// SIMATIC S7-200 SMART project (STEP 7-Micro/WIN SMART), CPU ST40

SYMBOL_TABLE USER1
Spa_vidé         V102.0   // Spa sans eau pour nettoyage
Compteur0        C0       // Compteur temps Brome
Compteur1        C1       // Compteur cycle filtration HORS usage spa
Compteur2        C2
Compteur3        C3       // Compteur cycle logo BROME
Compteur4        C4       // Compteur jours vérif brome
Bp_Dde_Jets      I0.0     // M/A jets
Bp_Dde_Air       I0.1     // M/A Turbine
Bp_Dde_Ecl       I0.2     // M/A Eclairage
Bp_Dde_Heater    I0.3     // M/A Chauffage=> Non utilisé depuis SPA
Bp_Mode_Hiver    I0.4     // Si=1 alors 1 cycle/jour
Filtration_Forcée I0.5     // Filtration forcée
Filtration_Auto  I0.6     // Filtration en auto
Bp_Arrêt         I0.7     // Arrêt des pompes
Symbol_140       M0.1     // Etat_Air
Bit_1            M1.0     // Forçage à 1
Symbol_28        M2.0     // ModBUS démarré
Symbol_25        M2.1     // carte n°1 ok
Symbol_26        M2.2     // carte n°2 ok
Symbol_27        M2.3     // carte n°3 ok
Symbol_85        M2.4     // carte n°4 ok
Bascule_SR_Jets  M10.0    // M/A jets
Symbol_49        M10.1    // Etat_Air
Bascule_SR_Air   M11.0    // M/A turbine
Bascule_SR_Ecl   M12.0    // M/A eclairage
Symbol_29        MB5      // Etat_Air
Symbol_83        MB10     // Etat_Air
Valeur_jets      MB16
Valeur_air       MB17
valeur_pac       MB18
Valeur_tampon    MB19
Pompe_Jets       Q0.0     // M/A Jets pompe
Pompe_Air        Q0.1     // M/A Turbine
Relais_Ecl       Q0.2     // M/A Eclairage
Relais_PAC       Q0.3     // M/A Pompe à chaleur SPA
Pompe_Filtration Q0.4     // M/A Pompe à filtration
Vanne_Remplissage Q0.5     // M/A Vanne remplissage
Fan_SSR          Q0.6     // Ventilateurs relais SSR et coffret
Led_Jets         Q1.0     // Led Bp Jets +5vdc
Led_Air          Q1.1     // Led Bp Air +5vdc
Led_Ecl          Q1.2     // Led Bp Ecl +5vdc
Led_Heat         Q1.3     // Led Bp Heat +5vdc
Led_Arret        Q1.4     // Led Bp Arrêt +5vdc
Led_Hiver        Q1.5     // Led Mode Hiver
TimerJets        T37      // Tempo jets 30 min
TimerAir         T38      // Tempo jets 30 min
TimerFilt        T39      // Tempo 54min
TimerCyc1        T40      // Tempo 54min
TimerCyc2        T41      // Tempo 54min
TimerCycFilt     T42
Bit_1Hz          T45
Symbol_45        T48      // Etat_Air
Bit_2Hz          T50
Symbol_137       T51      // Etat_Air
Symbol_134       T52      // Etat_Air
Symbol_44        T53      // Etat_Air
TimerRstTpsPompJets T54      // Timer reset tps marche pompe jets
TimerFillSpa     T55      // Timer Remplissage Spa
TimerCarte7      T56      // TimerCycleModbus carte7
TimerCarte6      T57      // TimerCycleModbus carte6
TimerCarte5      T58      // TimerCycleModbus carte5
TimerCycleModbus T59      // TimerCycleModbus
TimerCarte1      T60      // TimerCycleModbus carte1
TimerCarte2      T61      // TimerCycleModbus carte2
TimerCarte3      T62      // TimerCycleModbus carte3
TimerCarte4      T63      // TimerCycleModbus carte4
TimerCycleRS485  T255     // Temporisation cartes RS485
Symbol_2         V10.0    // Etat_Air
Symbol_3         V10.1    // Etat_Air
Symbol_8         V10.2    // Etat_Air
Symbol_0         V11.0    // Demande Air
Symbol_1         V11.1    // Etat_Air
Symbol_7         V11.2    // Etat_Air
Symbol_5         V12.0    // Etat_Air
Symbol_4         V12.1    // Etat_Air
Symbol_6         V12.2    // Etat_Air
DiminuerTauxpH   V51.1
AugmenterTauxpH  V51.2
pHOk             V51.3
Symbol_19        V70.0    // Etat_Air
Symbol_90        V101.0   // Etat_Air
Symbol_91        V201.0   // Etat_Air
BromeLogo        V702.0   // Demande vérification Brome
Symbol_88        V1220.0  // Etat_Air
Symbol_89        V1220.1  // Etat_Air
AckDef           V1510.0  // Effacement des défauts
ResetTpsPompeJets V1510.1  // RàZ du totaliseur de la pompe jets
Symbol_62        V1510.2  // Etat_Air
Symbol_135       V1510.3  // Etat_Air
Symbol_136       V1510.4  // Etat_Air
Symbol_138       V1510.5  // Etat_Air
ResetDéfBrome    V1510.6  // Etat_Air
CorrectionpH     V1799.3  // 1 cycle de correction du pH
Symbol_142       V6000.1  // Etat_Air
Symbol_143       V6000.2  // Etat_Air
Symbol_144       V6000.3  // Etat_Air
Symbol_145       V6000.4  // Etat_Air
Symbol_146       V6000.5  // Etat_Air
Symbol_39        VB0      // Etat_Air
Symbol_40        VB1      // Etat_Air
Symbol_38        VB2      // Etat_Air
Symbol_41        VB3      // Etat_Air
Symbol_56        VB4      // Etat_Air
Symbol_96        VB5      // Etat_Air
Symbol_9         VB15     // Etat_Air
Fond_écran_HMI   VB15
Symbol_11        VB100    // Etat_Air
Symbol_12        VB200    // Etat_Air
Symbol_48        VB500    // Etat_Air
EtatFiltration   VB600    // Etat filtration à sable/cartouche
Symbol_20        VB700    // Etat_Air
Symbol_13        VB1100   // Etat_Air
Symbol_51        VB1200   // Etat_Air
Symbol_92        VB1202   // Etat_Air
Symbol_74        VB1300   // Etat_Air
Symbol_14        VB1400   // Etat_Air
Symbol_93        VB1500   // Etat_Air
Symbol_141       VB1510   // Etat_Air
SensRotationPump VB1710   // 0: sens CW / 1: sens CCW
AccelRotationPump VB1711   // Accélération moteur pompe
Symbol_50        VB2000   // Etat_Air
Symbol_100       VB3000   // Etat_Air
Symbol_21        VD1000   // Etat_Air
NbreTrPump       VD1714   // Nombre tours pompe: 1tr=25600pts
VolumeInjection  VD1780   // Nombre tours injection
NbreTourPompeIhm VD1784   // Nombre tour pompe en manu
Tps_Mar_Pomp_Jets VD3000   // Tps_Mar_Pomp_Jets
Symbol_35        VD3004   // Etat_Air
Symbol_101       VD3008   // Etat_Air
Tps_Mar_Pomp_Air VD3010   // Tps_Mar_Pomp_Air
Symbol_103       VD3012   // Etat_Air
Symbol_15        VD3016   // Etat_Air
Tps_Mar_Pomp_Ecl VD3020   // Tps_Mar_Pomp_Ecl
Symbol_82        VD3028   // Etat_Air
Tps_Mar_Pomp_Pac VD3030   // Tps_Mar_Pomp_Pac
Symbol_63        VD3032   // Etat_Air
Symbol_64        VD3036   // Etat_Air
Tps_Mar_Pomp_Filt VD3040   // Tps_Mar_Pomp_Filt
Symbol_79        VD3044   // Etat_Air
Symbol_81        VD3048   // Etat_Air
Symbol_97        VD3052   // Etat_Air
Symbol_47        VD3100   // Etat_Air
Symbol_16        VD3104   // Etat_Air
Symbol_17        VD3108   // Etat_Air
Symbol_18        VD3112   // Etat_Air
Symbol_133       VD3116   // Etat_Air
Symbol_98        VD3120   // Etat_Air
Symbol_99        VD3124   // Etat_Air
Symbol_102       VD3128   // Etat_Air
Symbol_105       VD3132   // Etat_Air
Symbol_106       VD3136   // Etat_Air
Symbol_107       VD3140   // Etat_Air
Symbol_108       VD3144   // Etat_Air
Symbol_109       VD3148   // Etat_Air
Symbol_110       VD3152   // Etat_Air
Symbol_60        VD3200   // Etat_Air
Symbol_61        VD3300   // Etat_Air
Symbol_111       VD3312   // Etat_Air
Symbol_112       VD3316   // Etat_Air
Symbol_113       VD3320   // Etat_Air
Symbol_114       VD3324   // Etat_Air
Symbol_115       VD3328   // Etat_Air
Symbol_116       VD3332   // Etat_Air
Symbol_117       VD3336   // Etat_Air
Symbol_118       VD3340   // Etat_Air
Symbol_119       VD3344   // Etat_Air
Symbol_120       VD3348   // Etat_Air
Symbol_121       VD3352   // Etat_Air
Symbol_65        VD3400   // Etat_Air
Symbol_122       VD3412   // Etat_Air
Symbol_123       VD3416   // Etat_Air
Symbol_124       VD3420   // Etat_Air
Symbol_125       VD3424   // Etat_Air
Symbol_126       VD3428   // Etat_Air
Symbol_127       VD3432   // Etat_Air
Symbol_128       VD3436   // Etat_Air
Symbol_129       VD3440   // Etat_Air
Symbol_130       VD3444   // Etat_Air
Symbol_131       VD3448   // Etat_Air
Symbol_132       VD3452   // Etat_Air
Symbol_10        VD30012  // Etat_Air
Symbol_77        VD30444  //
NbreCycleFilt    VW7      // nombre cycle filtration par jour
LimiteFiltrationJour VW120    // LimiteFiltrationJour
Symbol_80        VW140    // Etat_Air
Symbol_78        VW150    // Etat_Air
Symbol_24        VW1000   // Temp_Eau
Symbol_30        VW1002   // Temp_Jets
Symbol_31        VW1004   // Temp_Air
Symbol_32        VW1006   // Temp_Filt
Symbol_33        VW1008   // Etat_Air
Symbol_34        VW1010   // Etat_Air
Symbol_37        VW1012   // Etat_Air
Symbol_36        VW1014   // Etat_Air
Symbol_43        VW1020   // Etat_Air
Symbol_46        VW1022   // Etat_Air
Symbol_58        VW1024   // Etat_Air
Symbol_59        VW1026   // Etat_Air
TempératureEau   VW1100   // Température Eau
Symbol_57        VW1102   // Température moteur Jets
Symbol_66        VW1104   // Température moteur Air
Symbol_67        VW1106   // Température moteur Filtration
Symbol_68        VW1108   //
Symbol_69        VW1110   //
Symbol_70        VW1112   //
Symbol_71        VW1114   //
Symbol_72        VW1120   //
Symbol_73        VW1122   //
Symbol_54        VW1200   // pH de l'eau
TauxpHBassin     VW1202   // Température de l'eau (pas utilisée)
LimitPhBas       VW1210   // Limite haute du pH
LimitPhHaut      VW1212   // Limite basse du pH
Symbol_75        VW1300   //
Symbol_76        VW1302   //
Symbol_86        VW1400   //
Symbol_87        VW1402   //
Symbol_94        VW1500   // Etat_Air
Symbol_95        VW1502   // Etat_Air
Demande_Remplissage_Spa VW1520   // Demande_Remplissage
VitesseRotationPump VW1712   // vitesse rotation pompe
TpsSurveillanceTauxpH VW1720   // Surveillance Taux pH toutes les 3h ou 12h
TpsSurveillancePhHiver VW1740   // TpsSurveillancePhHiver
TpsSurveillancePhEté VW1750   // TpsSurveillancePhEté
VitesseRotationPompe VW1770   // Vitesse rotation pompe pH
NombreTourPompe  VW1784   // Nombre tour pompe par défaut
ValeurInjectionDefaut VW1786   // valeur par défaut pour rester à 7.4
Symbol_52        VW2000   //
Symbol_53        VW2002   //
Symbol_22        VW3000   // Etat_Air
Symbol_104       VW3002   // Etat_Air
Symbol_23        VW3004   // Etat_Air
Symbol_84        VW3304   // Etat_Air
OffsetPh         VW7000   // offset sur sonde pH
OffsetOrp        VW7002   // Offset sonde ORP
END_SYMBOL_TABLE

SYMBOL_TABLE Table 2
PTO3_Status      SMB580   // PTO3 Status
PLS3_Ovr         SM580.6  // PTO3 pipeline overflow/underflow, loading pipeline while full or transferring an empty pipeline: 0=No overflow; 1=Pipeline overflow/underflow
PLS3_Idle        SM580.7  // PTO3 idle: 0 = PTO in progress;1= PTO is idle
PLS3_Ctrl        SMB581   // Monitor and control PTO3 (Pulse Train Output) and PWM3 (Pulse Width Modulation) for Q0.2
PLS3_Cycle_Update SM581.0  // PTO3/PWM3 update the cycle time or frequency value: 0=no update; 1=write new cycle time/frequency
PWM3_PW_Update   SM581.1  // PWM3 update the pulse width value: 0=no update; 1= write new pulse width
PTO3_PC_Update   SM581.2  // PTO3 update the pulse count value: 0=no update; 1= write new pulse count
PWM3_TimeBase    SM581.3  // PWM3 time base: 0=1us/tick, 1=1ms/tick
PLS3_Select      SM581.6  // PTO3/PWM3 mode select: 0=PWM; 1=PTO.
PLS3_Enable      SM581.7  // PTO3/PWM3 enable: 0=disable; 1=enable.
PLS3_Cycle       SMW582   // PWM3 cycle time value (2 to 65,535 units of time base); PTO3 frequency value (1 to 65,535 Hz)
PWM3_PW          SMW584   // PWM3 pulse width value (0 to 65,535 units of time base)
PTO3_PC          SMD586   // PTO3 pulse count value (1 to 2^32 - 1)
PLS3_Abort_AE    SM580.4  // PTO3 profile was aborted due to an add error: 0=no abort; 1=aborted
PLS3_Disable_UC  SM580.5  // PTO3 user manually disabled a PTO profile while it was running: 0=not disabled; 1=manually disabled
PTO3_Operation   SM581.5  // PTO3 select single/multiple segment operation: 0=single; 1=multiple
PTO3_Seg_Num     SMB590   // The currently executing segment number for PTO3's profile
PTO3_Profile_Offset SMW592   // Starting location of PTO3's profile table (byte offset from V0)
HSC0_TYPE        SMB195   // HSC0 type: 0=Count 1=Frequency
HSC0_FREQ_PERIOD SMB196   // HSC0 frequency measuring period: 0=1s 1=100ms 2=10ms
HSC1_TYPE        SMB197   // HSC1 type: 0=Count 1=Frequency
HSC1_FREQ_PERIOD SMB198   // HSC1 frequency measuring period: 0=1s 1=100ms 2=10ms
HSC2_TYPE        SMB199   // HSC2 type: 0=Count 1=Frequency
HSC2_FREQ_PERIOD SMB200   // HSC2 frequency measuring period: 0=1s 1=100ms 2=10ms
HSC3_TYPE        SMB201   // HSC3 type: 0=Count 1=Frequency
HSC3_FREQ_PERIOD SMB202   // HSC3 frequency measuring period: 0=1s 1=100ms 2=10ms
HSC4_TYPE        SMB203   // HSC4 type: 0=Count 1=Frequency
HSC4_FREQ_PERIOD SMB204   // HSC4 frequency measuring period: 0=1s 1=100ms 2=10ms
HSC5_TYPE        SMB205   // HSC5 type: 0=Count 1=Frequency
HSC5_FREQ_PERIOD SMB206   // HSC5 frequency measuring period: 0=1s 1=100ms 2=10ms
END_SYMBOL_TABLE

ORGANIZATION_BLOCK PPAL:OB1
TITLE=COMMENTAIRES DE PROGRAMME
VAR
Etat_Jets:BOOL;	// L0.0 Etat Jets
Sortie_Jets:BOOL;	// L0.1 Pilotage Sortie Jets
Voyant_Jets:BOOL;	// L0.2 Voyant +5vdc Jets
END_VAR
BEGIN
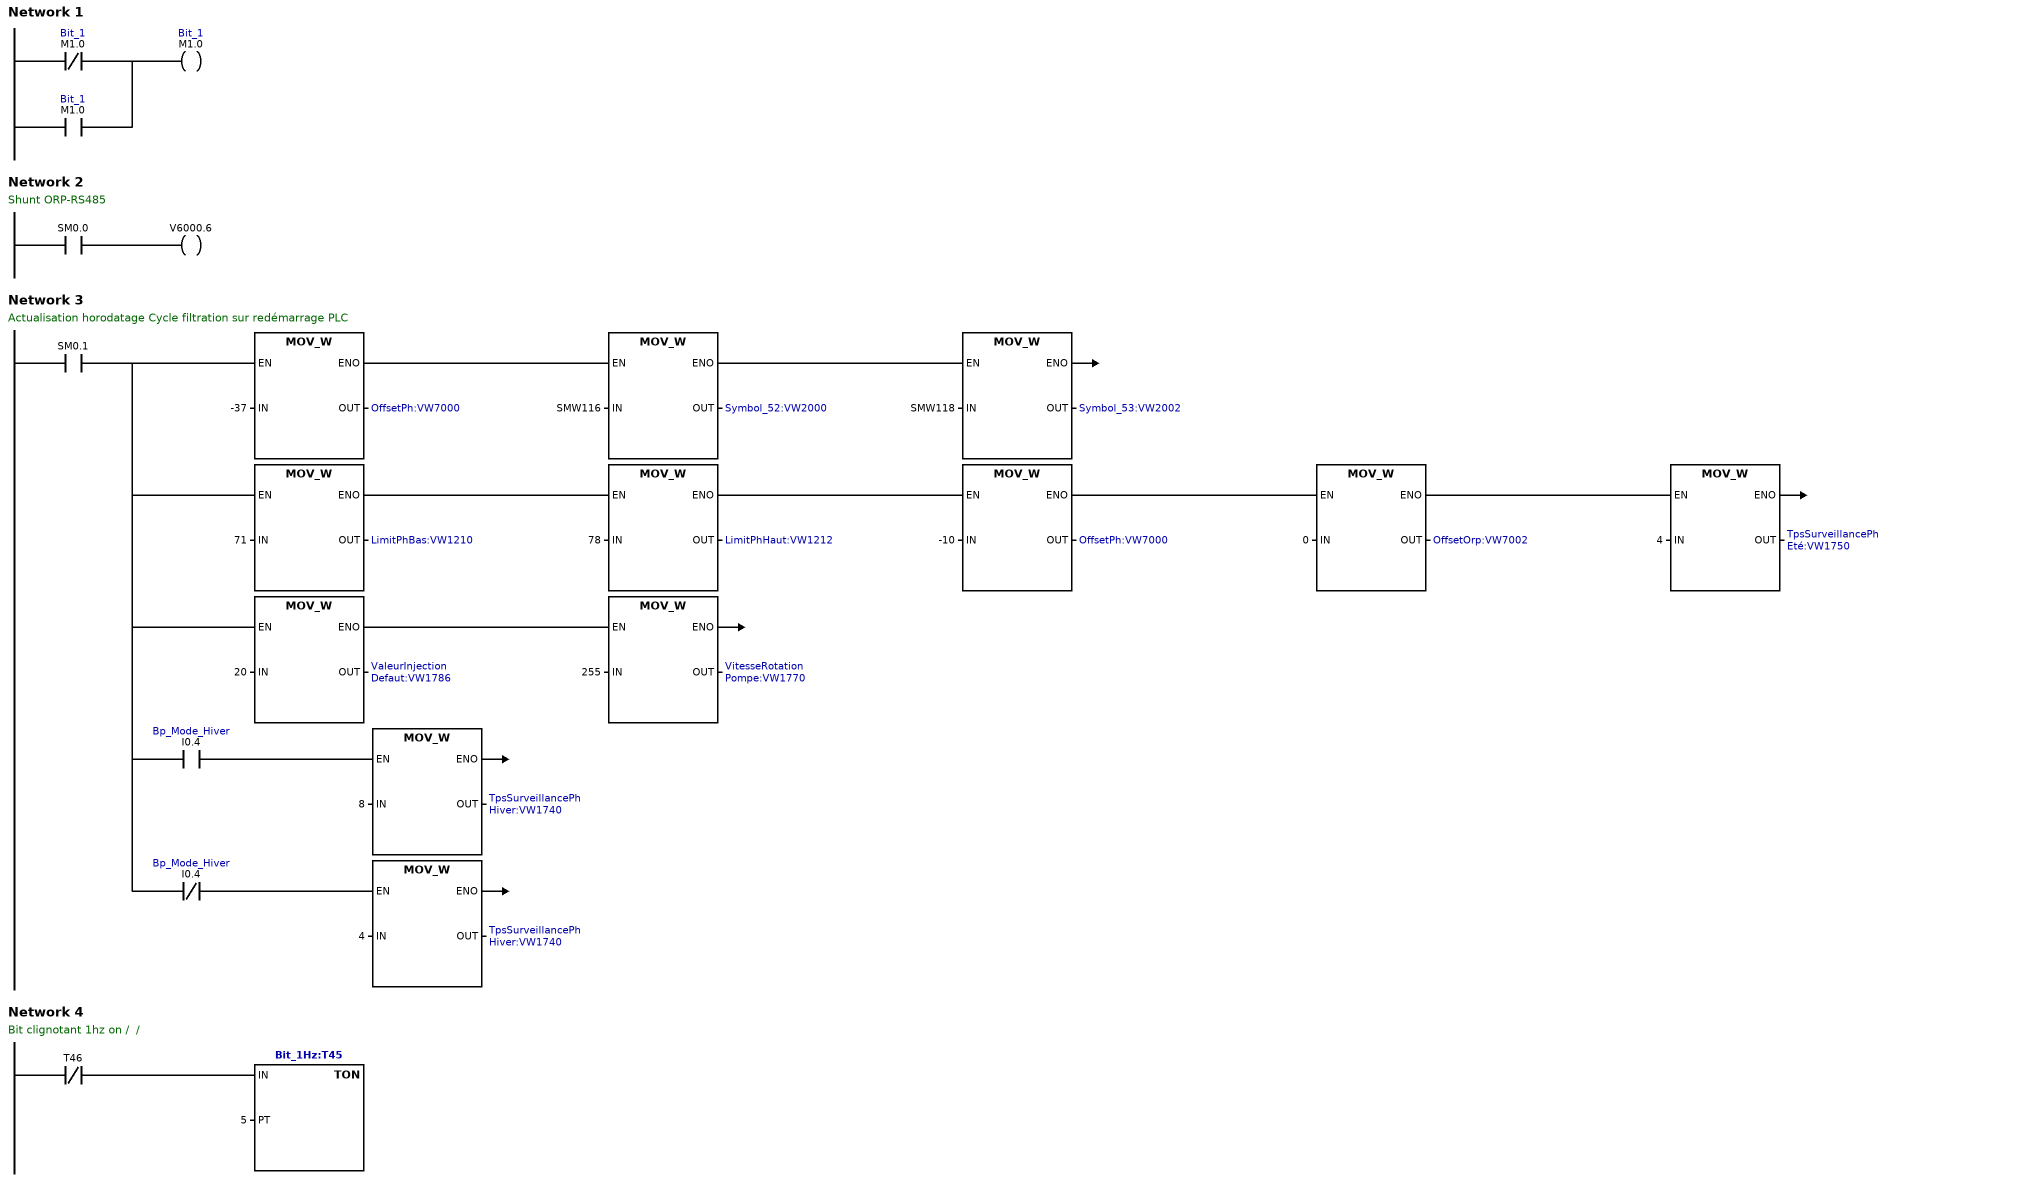
Network 1
LDN    Bit_1:M1.0
O      Bit_1:M1.0
=      Bit_1:M1.0
Network 2
// Shunt ORP-RS485
LD     SM0.0
=      V6000.6
Network 3
// Actualisation horodatage Cycle filtration sur redémarrage PLC
LD     SM0.1
LPS
MOVW   -37, OffsetPh:VW7000
AENO
MOVW   SMW116, Symbol_52:VW2000
AENO
MOVW   SMW118, Symbol_53:VW2002
LRD
MOVW   71, LimitPhBas:VW1210
AENO
MOVW   78, LimitPhHaut:VW1212
AENO
MOVW   -10, OffsetPh:VW7000
AENO
MOVW   0, OffsetOrp:VW7002
AENO
MOVW   4, TpsSurveillancePhEté:VW1750
LRD
MOVW   20, ValeurInjectionDefaut:VW1786
AENO
MOVW   255, VitesseRotationPompe:VW1770
LRD
A      Bp_Mode_Hiver:I0.4
MOVW   8, TpsSurveillancePhHiver:VW1740
LPP
AN     Bp_Mode_Hiver:I0.4
MOVW   4, TpsSurveillancePhHiver:VW1740
Network 4
// Bit clignotant 1hz on
// 
// 
LDN    T46
TON    Bit_1Hz:T45, 5
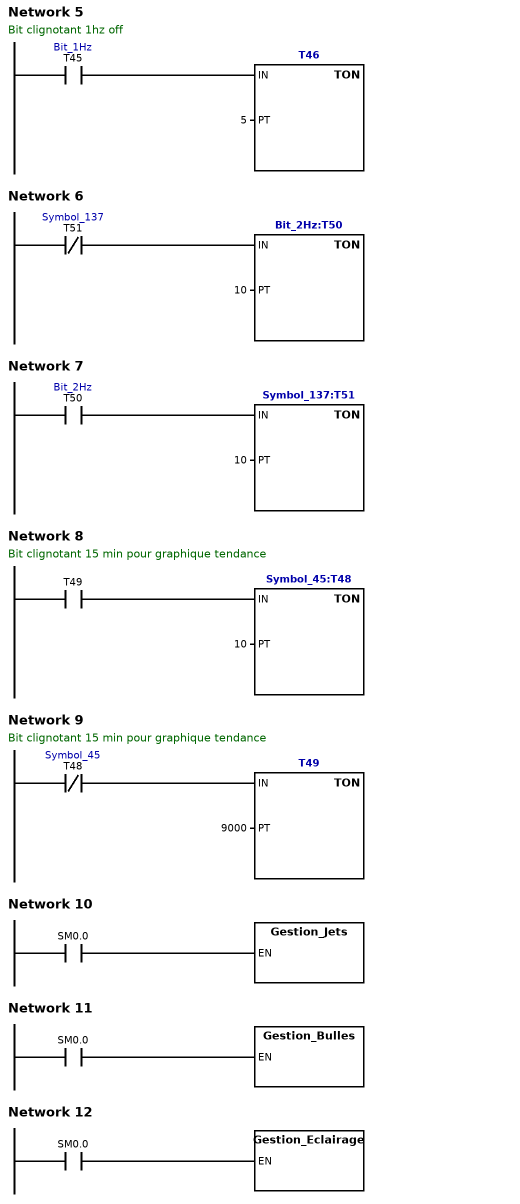
Network 5
// Bit clignotant 1hz off
LD     Bit_1Hz:T45
TON    T46, 5
Network 6
LDN    Symbol_137:T51
TON    Bit_2Hz:T50, 10
Network 7
LD     Bit_2Hz:T50
TON    Symbol_137:T51, 10
Network 8
// Bit clignotant 15 min pour graphique tendance
LD     T49
TON    Symbol_45:T48, 10
Network 9
// Bit clignotant 15 min pour graphique tendance
LDN    Symbol_45:T48
TON    T49, 9000
Network 10
LD     SM0.0
CALL   Gestion_Jets:SBR0
Network 11
LD     SM0.0
CALL   Gestion_Bulles:SBR1
Network 12
LD     SM0.0
CALL   Gestion_Eclairage:SBR2
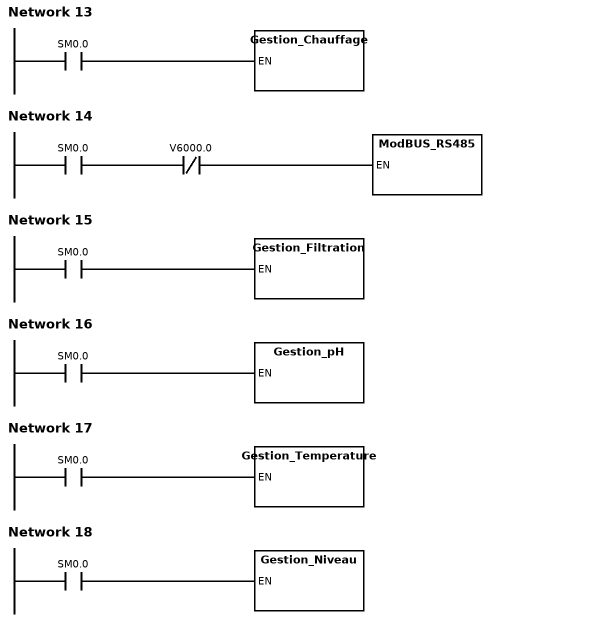
Network 13
LD     SM0.0
CALL   Gestion_Chauffage:SBR3
Network 14
LD     SM0.0
AN     V6000.0
CALL   ModBUS_RS485:SBR5
Network 15
LD     SM0.0
CALL   Gestion_Filtration:SBR7
Network 16
LD     SM0.0
CALL   Gestion_pH:SBR4
Network 17
LD     SM0.0
CALL   Gestion_Temperature:SBR6
Network 18
LD     SM0.0
CALL   Gestion_Niveau:SBR14
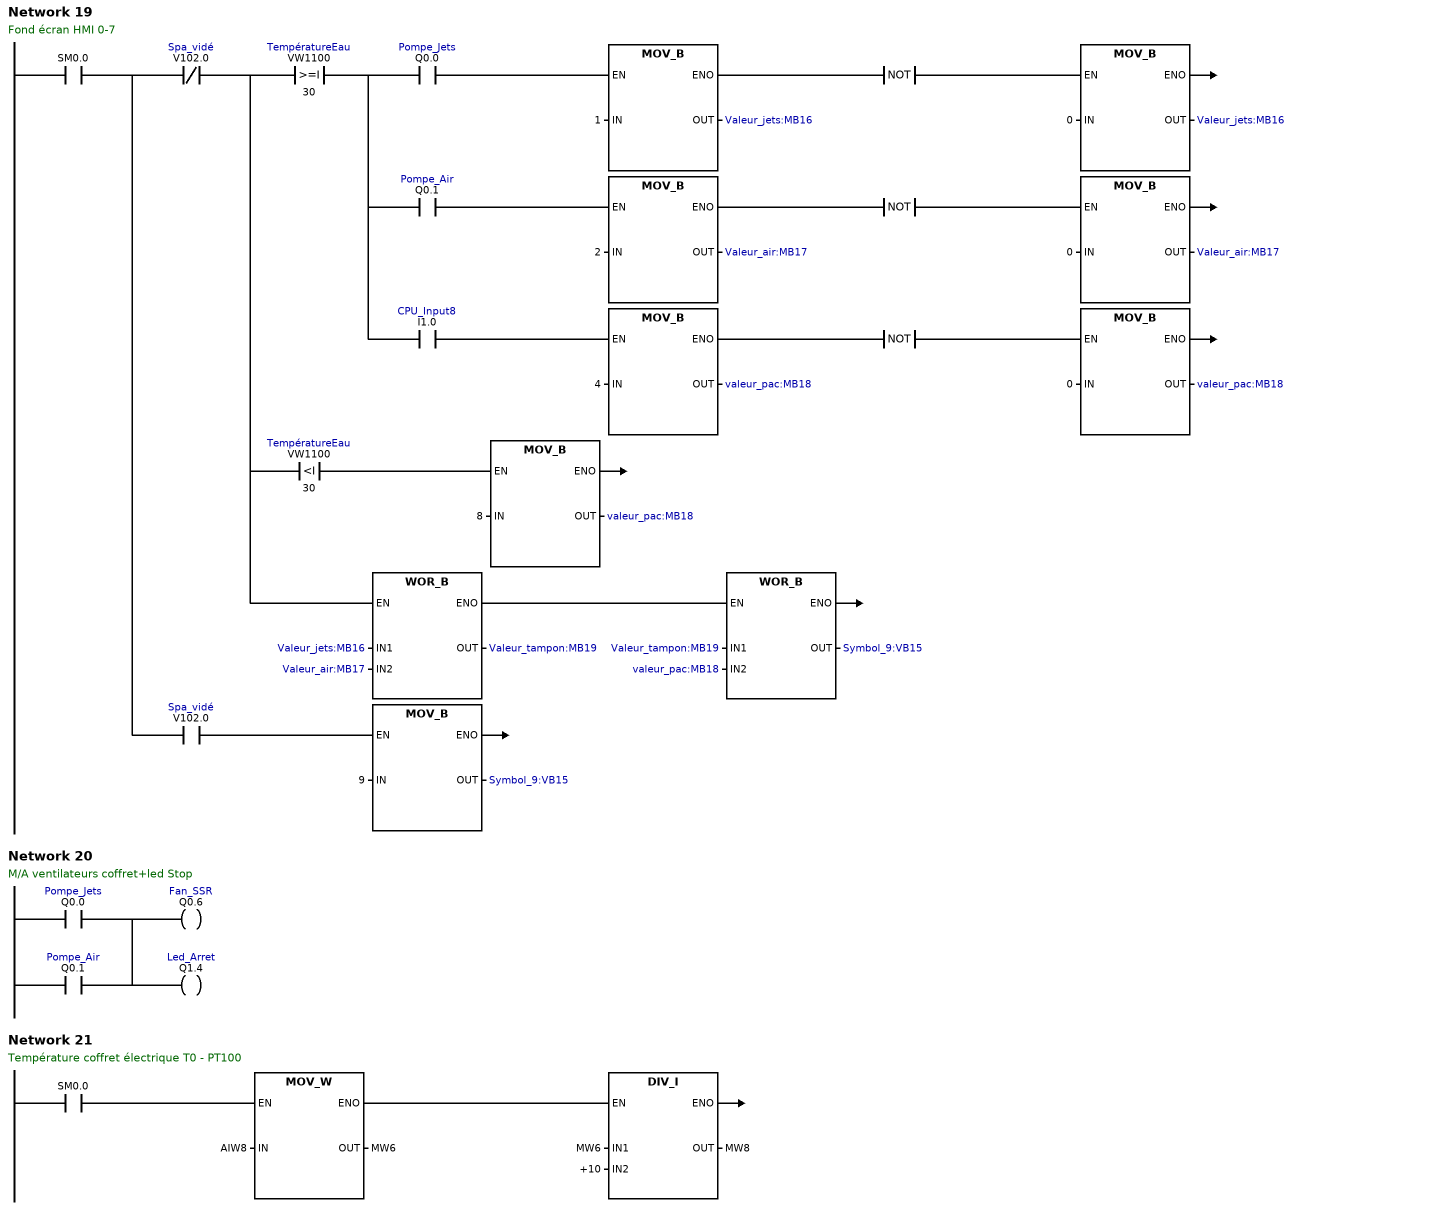
Network 19
// Fond écran HMI 0-7
LD     SM0.0
LPS
AN     Spa_vidé:V102.0
LPS
AW>=   TempératureEau:VW1100, 30
LPS
A      Pompe_Jets:Q0.0
MOVB   1, Valeur_jets:MB16
AENO
NOT
MOVB   0, Valeur_jets:MB16
LRD
A      Pompe_Air:Q0.1
MOVB   2, Valeur_air:MB17
AENO
NOT
MOVB   0, Valeur_air:MB17
LPP
A      CPU_Input8:I1.0
MOVB   4, valeur_pac:MB18
AENO
NOT
MOVB   0, valeur_pac:MB18
LPP
LPS
AW<    TempératureEau:VW1100, 30
MOVB   8, valeur_pac:MB18
LPP
MOVB   Valeur_jets:MB16, Valeur_tampon:MB19
AENO
ORB    Valeur_air:MB17, Valeur_tampon:MB19
AENO
MOVB   Valeur_tampon:MB19, Symbol_9:VB15
ORB    valeur_pac:MB18, Symbol_9:VB15
LPP
A      Spa_vidé:V102.0
MOVB   9, Symbol_9:VB15
Network 20
// M/A ventilateurs coffret+led Stop
LD     Pompe_Jets:Q0.0
O      Pompe_Air:Q0.1
=      Fan_SSR:Q0.6
=      Led_Arret:Q1.4
Network 21
// Température coffret électrique T0 - PT100
LD     SM0.0
MOVW   AIW8, MW6
AENO
MOVW   MW6, MW8
/I     +10, MW8
END_ORGANIZATION_BLOCK

SUBROUTINE_BLOCK Gestion_Jets:SBR0
TITLE=COMMENTAIRES DE SOUS-PROGRAMME
VAR
Etat_Jets:BOOL;	// L0.0 
END_VAR
BEGIN
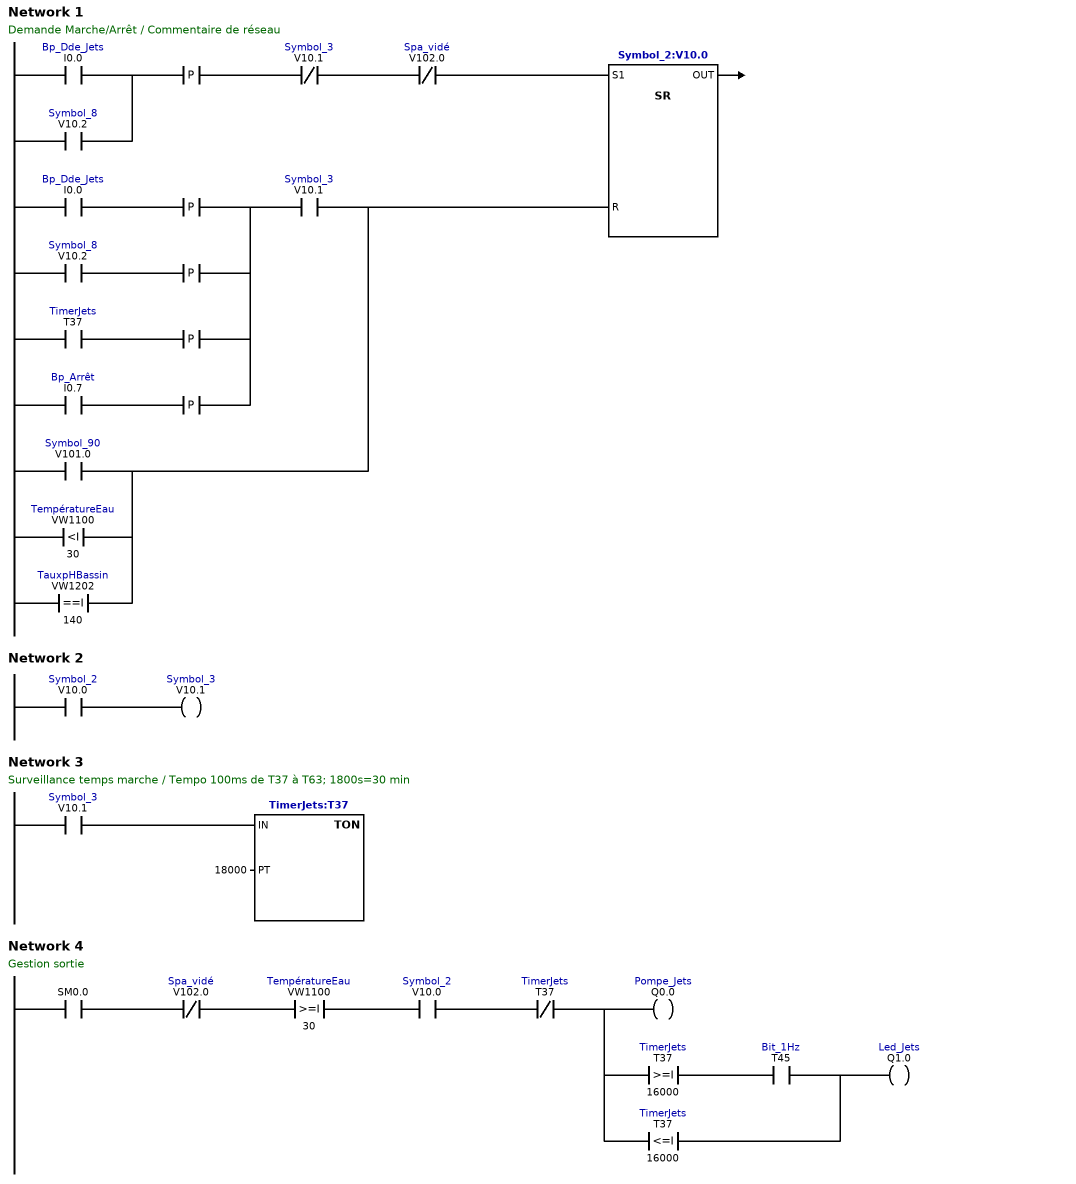
Network 1
// Demande Marche/Arrêt
// Commentaire de réseau
LD     Bp_Dde_Jets:I0.0
O      Symbol_8:V10.2
EU
AN     Symbol_3:V10.1
AN     Spa_vidé:V102.0
LD     Bp_Dde_Jets:I0.0
EU
LD     Symbol_8:V10.2
EU
OLD
LD     TimerJets:T37
EU
OLD
LD     Bp_Arrêt:I0.7
EU
OLD
A      Symbol_3:V10.1
LD     Symbol_90:V101.0
OW<    TempératureEau:VW1100, 30
OW=    TauxpHBassin:VW1202, 140
OLD
NOT
A      Symbol_2:V10.0
OLD
=      Symbol_2:V10.0
Network 2
LD     Symbol_2:V10.0
=      Symbol_3:V10.1
Network 3
// Surveillance temps marche
// Tempo 100ms de T37 à T63; 1800s=30 min
LD     Symbol_3:V10.1
TON    TimerJets:T37, 18000
Network 4
// Gestion sortie
LD     SM0.0
AN     Spa_vidé:V102.0
AW>=   TempératureEau:VW1100, 30
A      Symbol_2:V10.0
AN     TimerJets:T37
=      Pompe_Jets:Q0.0
LDW>=  TimerJets:T37, 16000
A      Bit_1Hz:T45
OW<=   TimerJets:T37, 16000
ALD
=      Led_Jets:Q1.0
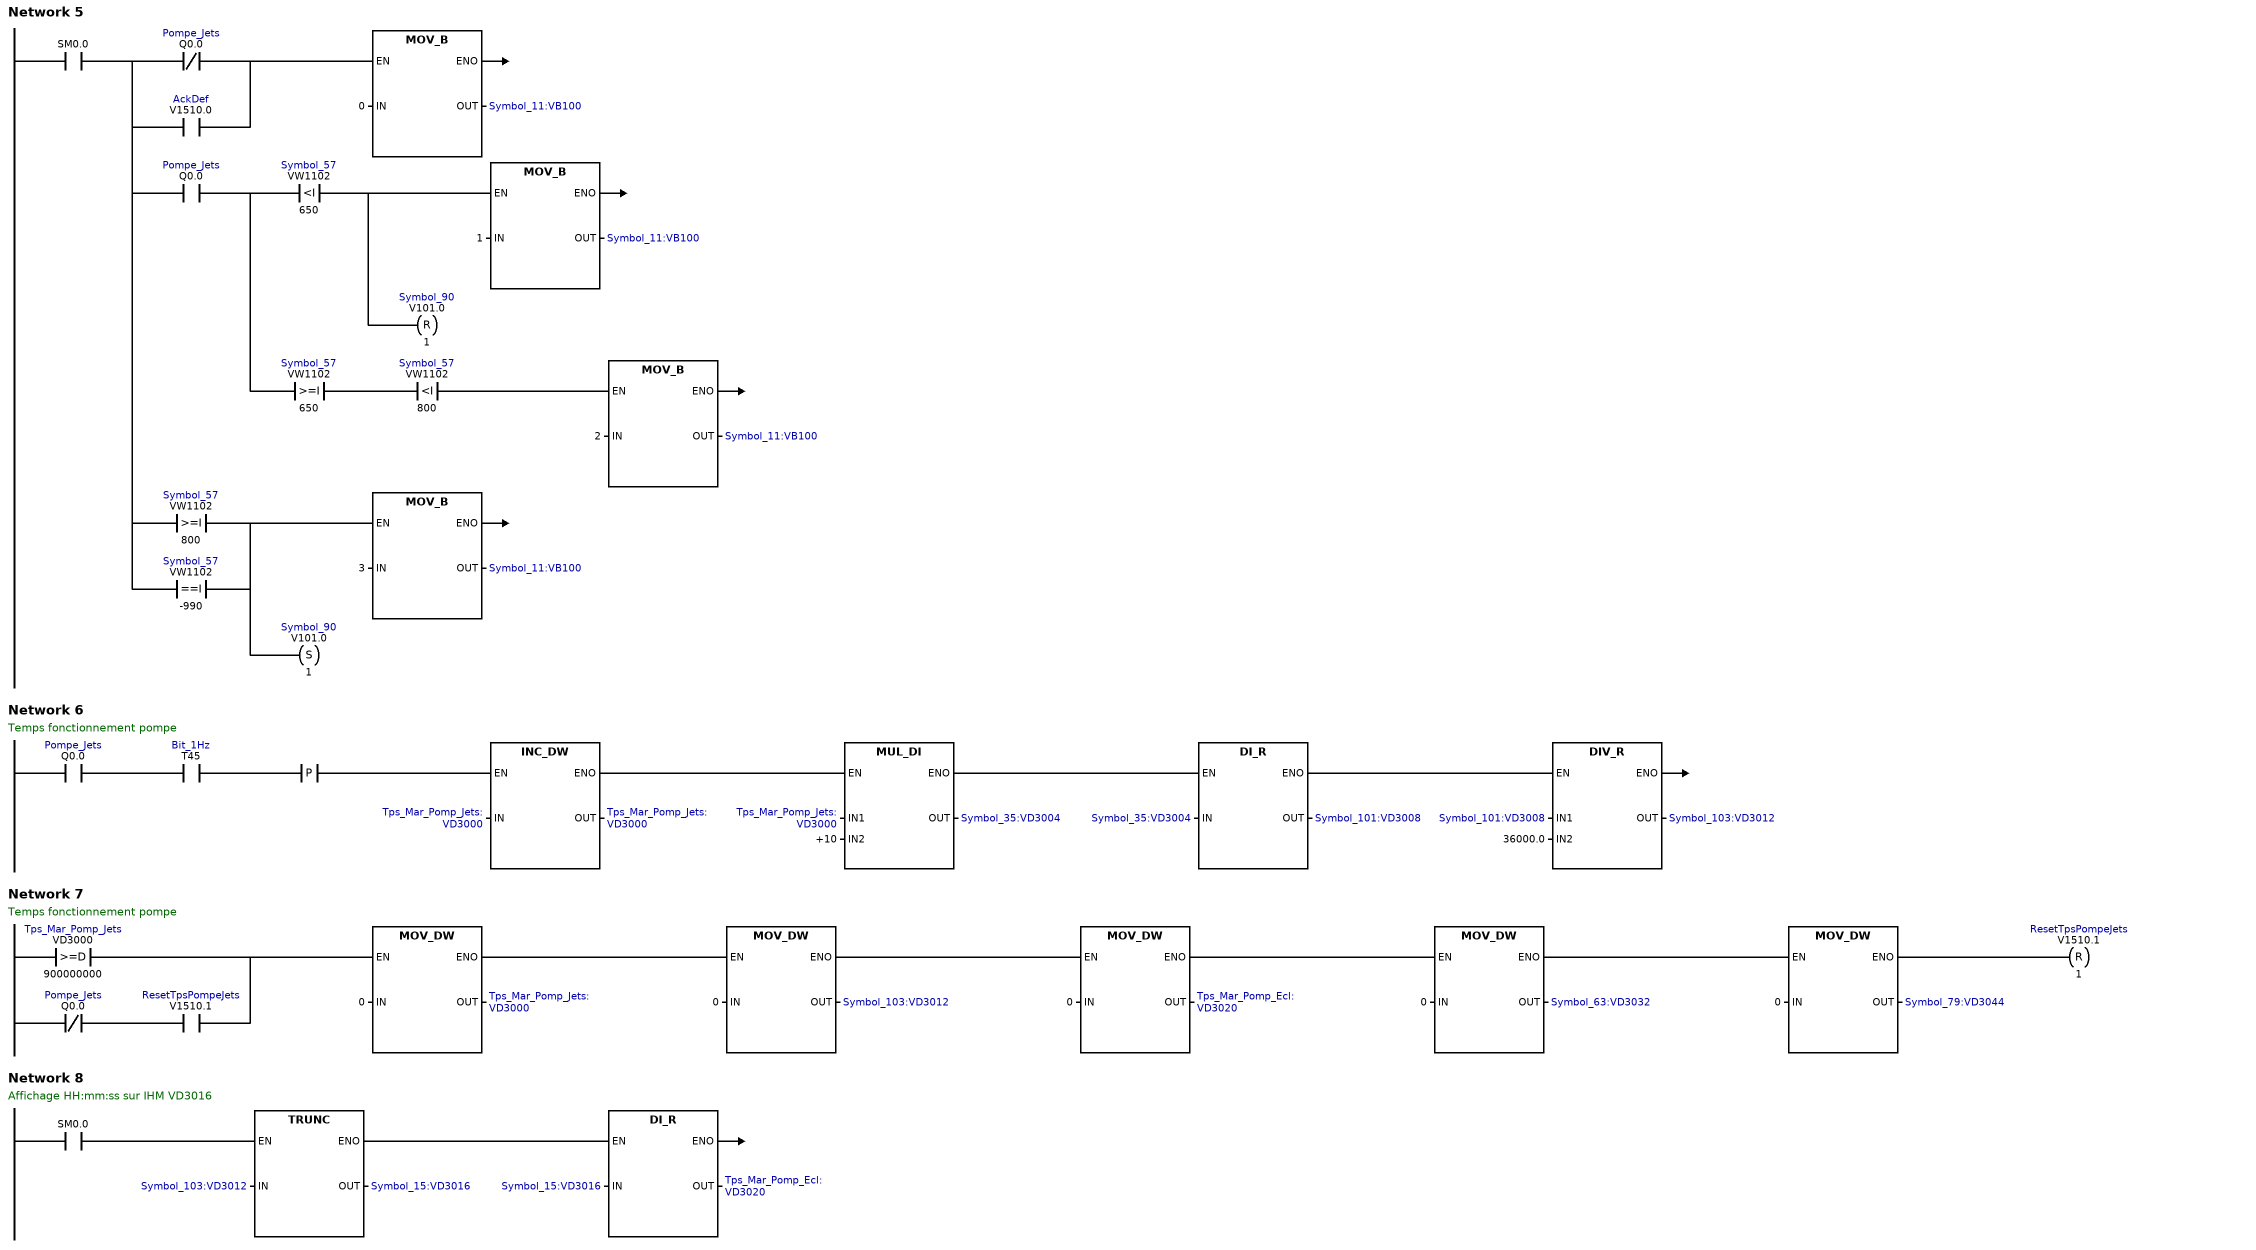
Network 5
LD     SM0.0
LPS
LDN    Pompe_Jets:Q0.0
O      AckDef:V1510.0
ALD
MOVB   0, Symbol_11:VB100
LRD
A      Pompe_Jets:Q0.0
LPS
AW<    Symbol_57:VW1102, 650
MOVB   1, Symbol_11:VB100
R      Symbol_90:V101.0, 1
LPP
AW>=   Symbol_57:VW1102, 650
AW<    Symbol_57:VW1102, 800
MOVB   2, Symbol_11:VB100
LPP
LDW>=  Symbol_57:VW1102, 800
OW=    Symbol_57:VW1102, -990
ALD
MOVB   3, Symbol_11:VB100
S      Symbol_90:V101.0, 1
Network 6
// Temps fonctionnement pompe
LD     Pompe_Jets:Q0.0
A      Bit_1Hz:T45
EU
INCD   Tps_Mar_Pomp_Jets:VD3000
AENO
MOVD   Tps_Mar_Pomp_Jets:VD3000, Symbol_35:VD3004
AENO
*D     +10, Symbol_35:VD3004
AENO
DTR    Symbol_35:VD3004, Symbol_101:VD3008
AENO
MOVR   Symbol_101:VD3008, Symbol_103:VD3012
/R     36000.0, Symbol_103:VD3012
Network 7
// Temps fonctionnement pompe
LDD>=  Tps_Mar_Pomp_Jets:VD3000, 900000000
LDN    Pompe_Jets:Q0.0
A      ResetTpsPompeJets:V1510.1
OLD
MOVD   0, Tps_Mar_Pomp_Jets:VD3000
AENO
MOVD   0, Symbol_103:VD3012
AENO
MOVD   0, Tps_Mar_Pomp_Ecl:VD3020
AENO
MOVD   0, Symbol_63:VD3032
AENO
MOVD   0, Symbol_79:VD3044
AENO
R      ResetTpsPompeJets:V1510.1, 1
Network 8
// Affichage HH:mm:ss sur IHM VD3016
LD     SM0.0
TRUNC  Symbol_103:VD3012, Symbol_15:VD3016
AENO
DTR    Symbol_15:VD3016, Tps_Mar_Pomp_Ecl:VD3020
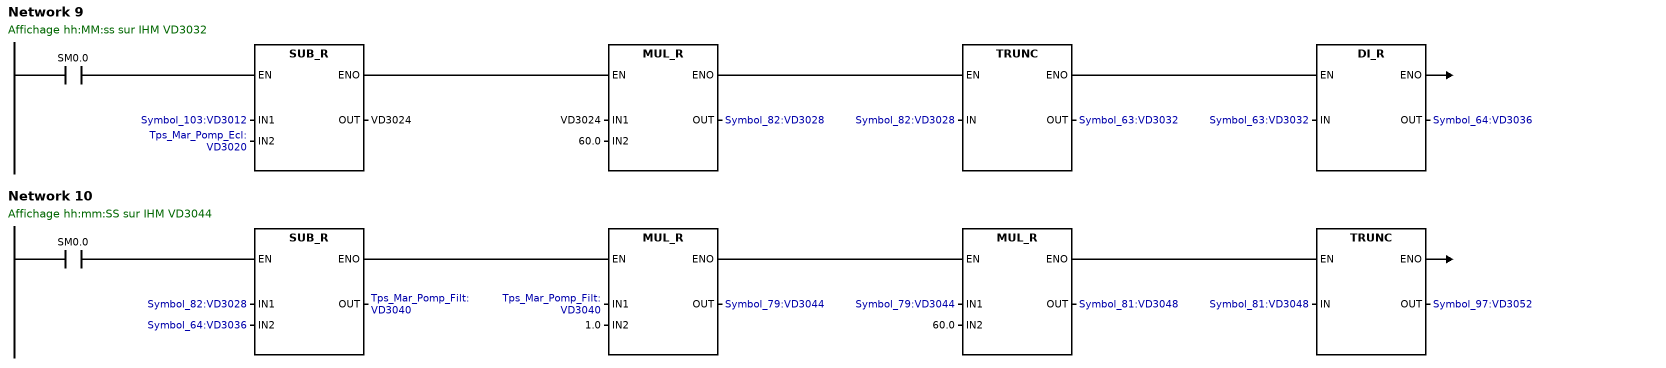
Network 9
// Affichage hh:MM:ss sur IHM VD3032
LD     SM0.0
MOVR   Symbol_103:VD3012, VD3024
AENO
-R     Tps_Mar_Pomp_Ecl:VD3020, VD3024
AENO
MOVR   VD3024, Symbol_82:VD3028
AENO
*R     60.0, Symbol_82:VD3028
AENO
TRUNC  Symbol_82:VD3028, Symbol_63:VD3032
AENO
DTR    Symbol_63:VD3032, Symbol_64:VD3036
Network 10
// Affichage hh:mm:SS sur IHM VD3044
LD     SM0.0
MOVR   Symbol_82:VD3028, Tps_Mar_Pomp_Filt:VD3040
AENO
-R     Symbol_64:VD3036, Tps_Mar_Pomp_Filt:VD3040
AENO
MOVR   Tps_Mar_Pomp_Filt:VD3040, Symbol_79:VD3044
AENO
*R     1.0, Symbol_79:VD3044
AENO
MOVR   Symbol_79:VD3044, Symbol_81:VD3048
AENO
*R     60.0, Symbol_81:VD3048
AENO
TRUNC  Symbol_81:VD3048, Symbol_97:VD3052
END_SUBROUTINE_BLOCK

SUBROUTINE_BLOCK Gestion_Bulles:SBR1
TITLE=COMMENTAIRES DE SOUS-PROGRAMME
VAR
Etat_Air:BOOL;	// L0.0 
END_VAR
BEGIN
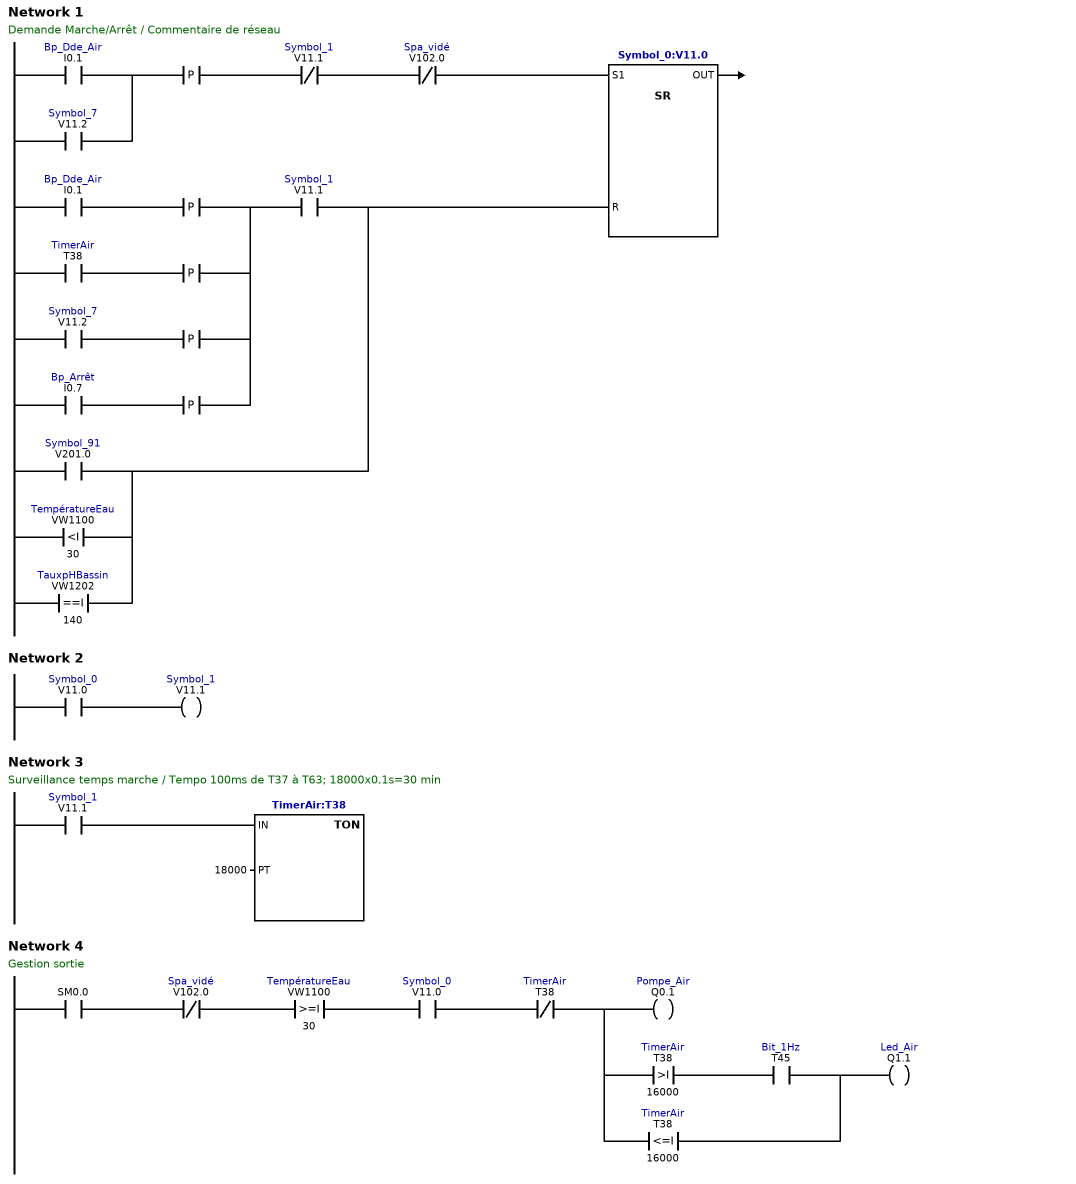
Network 1
// Demande Marche/Arrêt
// Commentaire de réseau
LD     Bp_Dde_Air:I0.1
O      Symbol_7:V11.2
EU
AN     Symbol_1:V11.1
AN     Spa_vidé:V102.0
LD     Bp_Dde_Air:I0.1
EU
LD     TimerAir:T38
EU
OLD
LD     Symbol_7:V11.2
EU
OLD
LD     Bp_Arrêt:I0.7
EU
OLD
A      Symbol_1:V11.1
LD     Symbol_91:V201.0
OW<    TempératureEau:VW1100, 30
OW=    TauxpHBassin:VW1202, 140
OLD
NOT
A      Symbol_0:V11.0
OLD
=      Symbol_0:V11.0
Network 2
LD     Symbol_0:V11.0
=      Symbol_1:V11.1
Network 3
// Surveillance temps marche
// Tempo 100ms de T37 à T63; 18000x0.1s=30 min
LD     Symbol_1:V11.1
TON    TimerAir:T38, 18000
Network 4
// Gestion sortie
LD     SM0.0
AN     Spa_vidé:V102.0
AW>=   TempératureEau:VW1100, 30
A      Symbol_0:V11.0
AN     TimerAir:T38
=      Pompe_Air:Q0.1
LDW>   TimerAir:T38, 16000
A      Bit_1Hz:T45
OW<=   TimerAir:T38, 16000
ALD
=      Led_Air:Q1.1
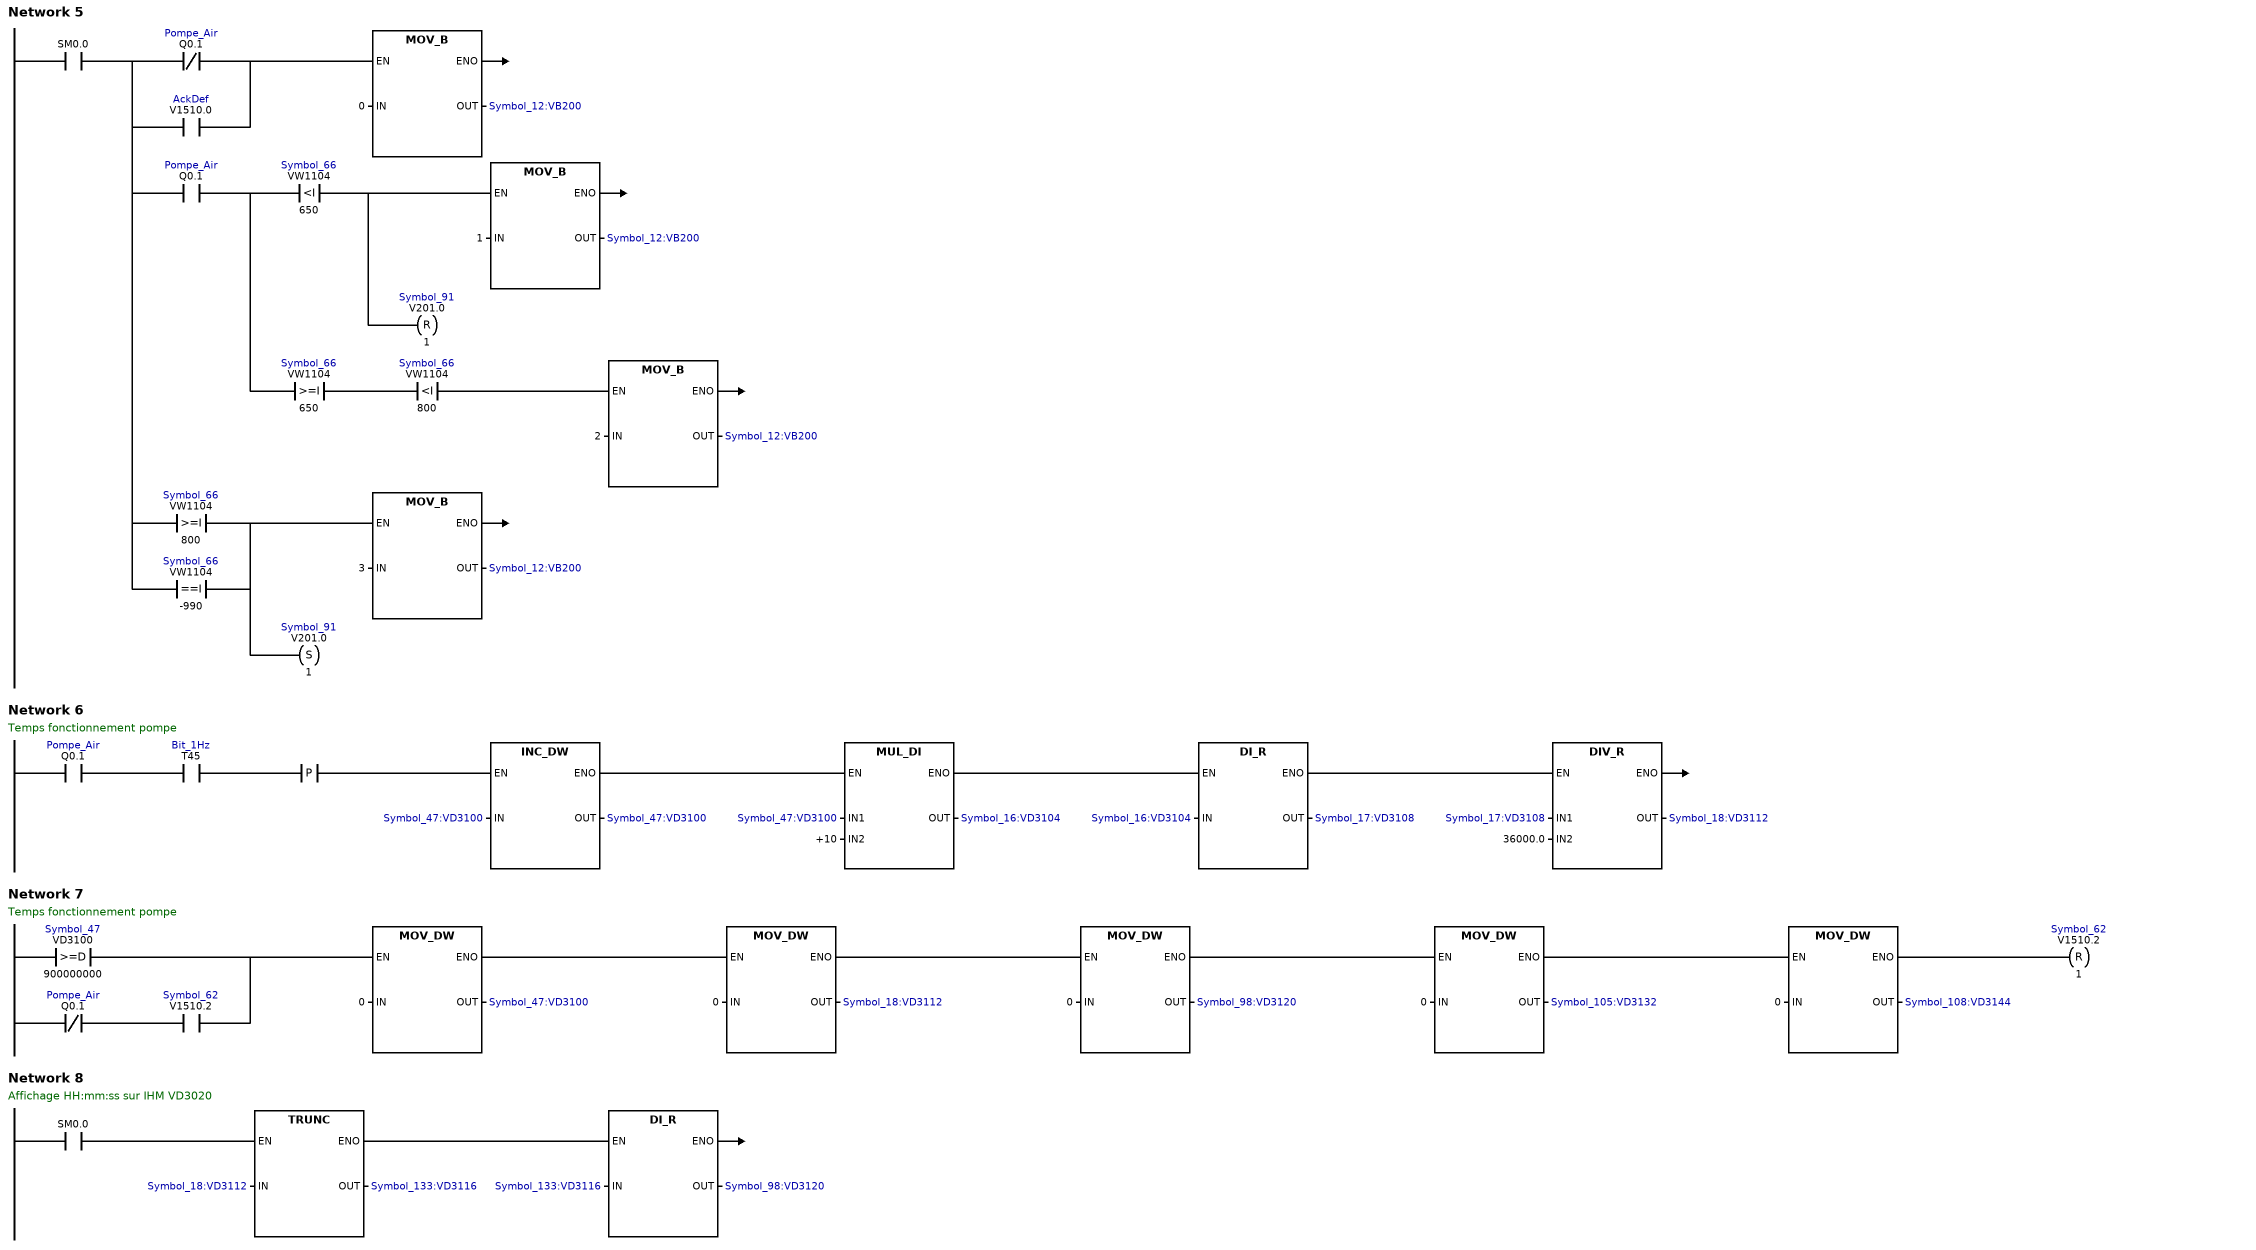
Network 5
LD     SM0.0
LPS
LDN    Pompe_Air:Q0.1
O      AckDef:V1510.0
ALD
MOVB   0, Symbol_12:VB200
LRD
A      Pompe_Air:Q0.1
LPS
AW<    Symbol_66:VW1104, 650
MOVB   1, Symbol_12:VB200
R      Symbol_91:V201.0, 1
LPP
AW>=   Symbol_66:VW1104, 650
AW<    Symbol_66:VW1104, 800
MOVB   2, Symbol_12:VB200
LPP
LDW>=  Symbol_66:VW1104, 800
OW=    Symbol_66:VW1104, -990
ALD
MOVB   3, Symbol_12:VB200
S      Symbol_91:V201.0, 1
Network 6
// Temps fonctionnement pompe
LD     Pompe_Air:Q0.1
A      Bit_1Hz:T45
EU
INCD   Symbol_47:VD3100
AENO
MOVD   Symbol_47:VD3100, Symbol_16:VD3104
AENO
*D     +10, Symbol_16:VD3104
AENO
DTR    Symbol_16:VD3104, Symbol_17:VD3108
AENO
MOVR   Symbol_17:VD3108, Symbol_18:VD3112
/R     36000.0, Symbol_18:VD3112
Network 7
// Temps fonctionnement pompe
LDD>=  Symbol_47:VD3100, 900000000
LDN    Pompe_Air:Q0.1
A      Symbol_62:V1510.2
OLD
MOVD   0, Symbol_47:VD3100
AENO
MOVD   0, Symbol_18:VD3112
AENO
MOVD   0, Symbol_98:VD3120
AENO
MOVD   0, Symbol_105:VD3132
AENO
MOVD   0, Symbol_108:VD3144
AENO
R      Symbol_62:V1510.2, 1
Network 8
// Affichage HH:mm:ss sur IHM VD3020
LD     SM0.0
TRUNC  Symbol_18:VD3112, Symbol_133:VD3116
AENO
DTR    Symbol_133:VD3116, Symbol_98:VD3120
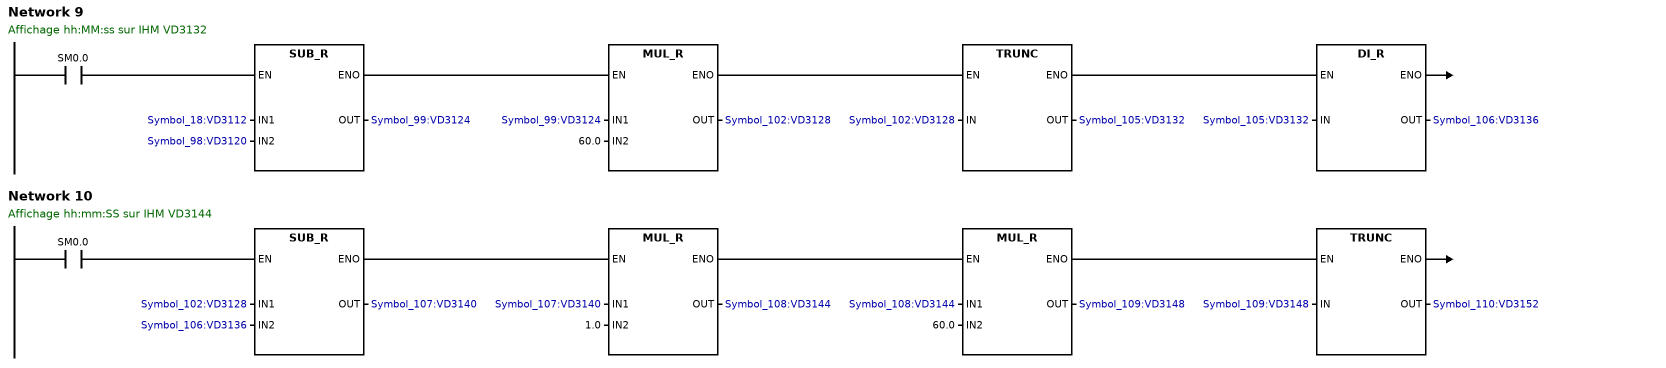
Network 9
// Affichage hh:MM:ss sur IHM VD3132
LD     SM0.0
MOVR   Symbol_18:VD3112, Symbol_99:VD3124
AENO
-R     Symbol_98:VD3120, Symbol_99:VD3124
AENO
MOVR   Symbol_99:VD3124, Symbol_102:VD3128
AENO
*R     60.0, Symbol_102:VD3128
AENO
TRUNC  Symbol_102:VD3128, Symbol_105:VD3132
AENO
DTR    Symbol_105:VD3132, Symbol_106:VD3136
Network 10
// Affichage hh:mm:SS sur IHM VD3144
LD     SM0.0
MOVR   Symbol_102:VD3128, Symbol_107:VD3140
AENO
-R     Symbol_106:VD3136, Symbol_107:VD3140
AENO
MOVR   Symbol_107:VD3140, Symbol_108:VD3144
AENO
*R     1.0, Symbol_108:VD3144
AENO
MOVR   Symbol_108:VD3144, Symbol_109:VD3148
AENO
*R     60.0, Symbol_109:VD3148
AENO
TRUNC  Symbol_109:VD3148, Symbol_110:VD3152
Network 13
// Titre de réseau
// Commentaire de réseau
END_SUBROUTINE_BLOCK

SUBROUTINE_BLOCK Gestion_Eclairage:SBR2
TITLE=COMMENTAIRES DE SOUS-PROGRAMME
VAR
Etat_Ecl:BOOL;	// L0.0 
END_VAR
BEGIN
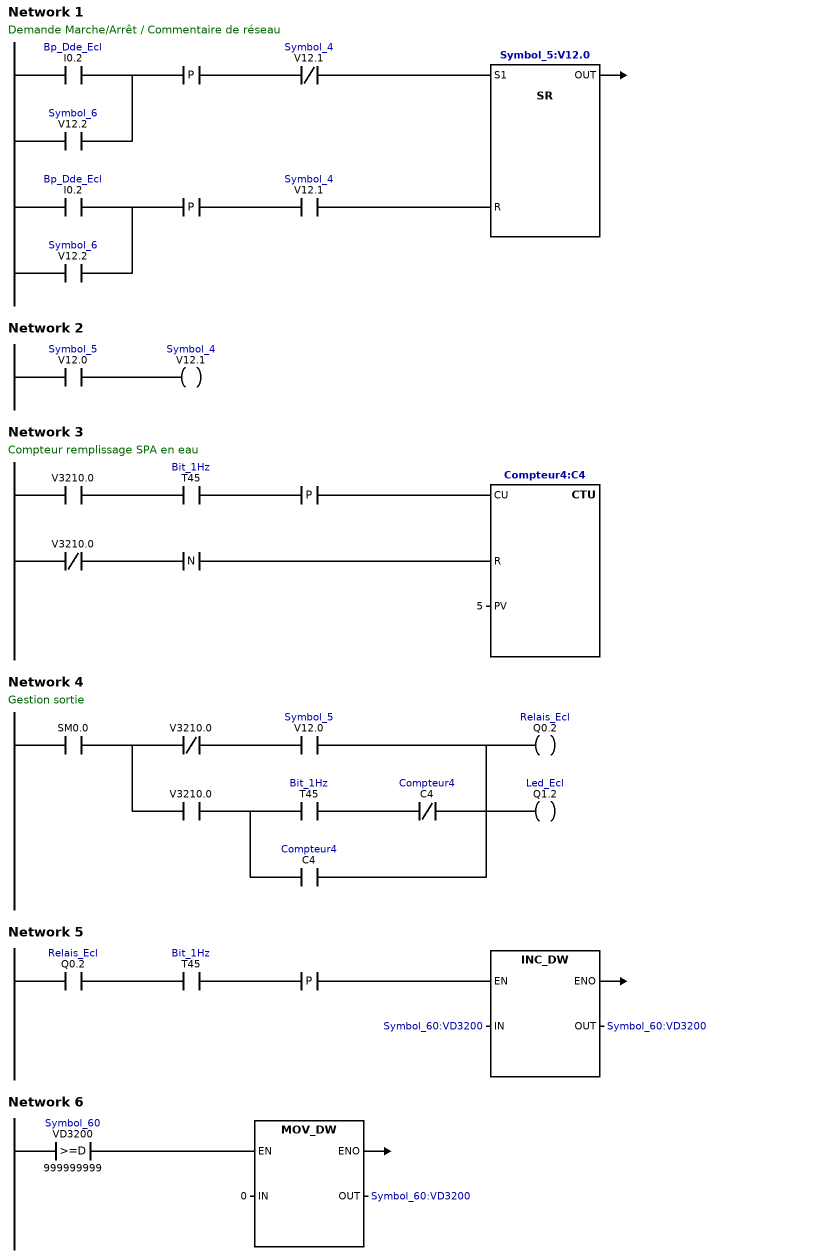
Network 1
// Demande Marche/Arrêt
// Commentaire de réseau
LD     Bp_Dde_Ecl:I0.2
O      Symbol_6:V12.2
EU
AN     Symbol_4:V12.1
LD     Bp_Dde_Ecl:I0.2
O      Symbol_6:V12.2
EU
A      Symbol_4:V12.1
NOT
A      Symbol_5:V12.0
OLD
=      Symbol_5:V12.0
Network 2
LD     Symbol_5:V12.0
=      Symbol_4:V12.1
Network 3
// Compteur remplissage SPA en eau
LD     V3210.0
A      Bit_1Hz:T45
EU
LDN    V3210.0
ED
CTU    Compteur4:C4, 5
Network 4
// Gestion sortie
LD     SM0.0
LDN    V3210.0
A      Symbol_5:V12.0
LD     V3210.0
LD     Bit_1Hz:T45
AN     Compteur4:C4
O      Compteur4:C4
ALD
OLD
ALD
=      Relais_Ecl:Q0.2
=      Led_Ecl:Q1.2
Network 5
LD     Relais_Ecl:Q0.2
A      Bit_1Hz:T45
EU
INCD   Symbol_60:VD3200
Network 6
LDD>=  Symbol_60:VD3200, 999999999
MOVD   0, Symbol_60:VD3200
Network 13
// Titre de réseau
// Commentaire de réseau
Network 23
// Titre de réseau
// Commentaire de réseau
END_SUBROUTINE_BLOCK

SUBROUTINE_BLOCK Gestion_Chauffage:SBR3
TITLE=COMMENTAIRES DE SOUS-PROGRAMME
BEGIN
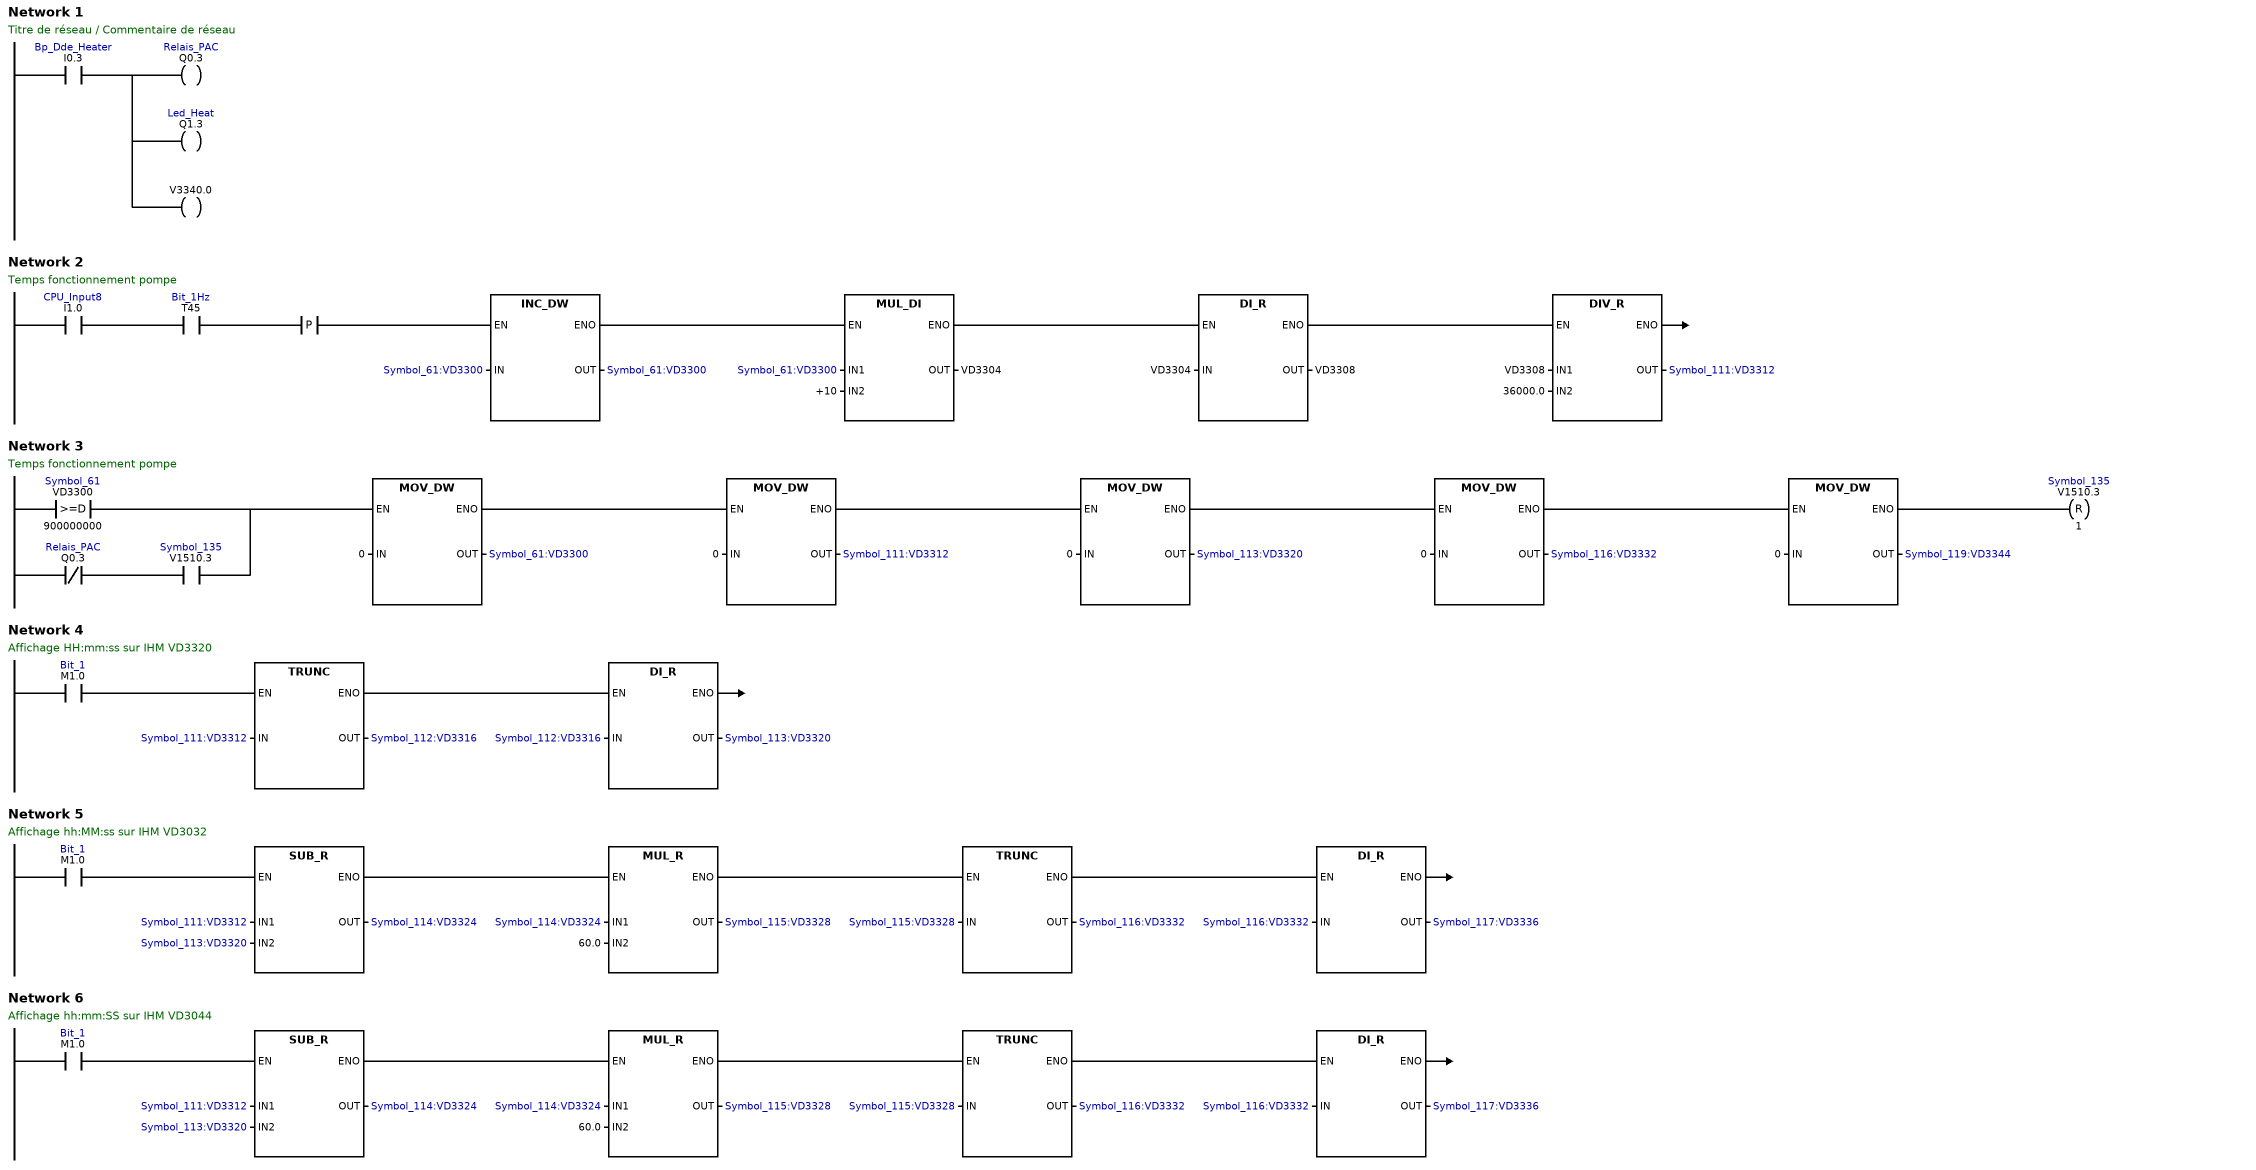
Network 1
// Titre de réseau
// Commentaire de réseau
LD     Bp_Dde_Heater:I0.3
=      Relais_PAC:Q0.3
=      Led_Heat:Q1.3
=      V3340.0
Network 2
// Temps fonctionnement pompe
LD     CPU_Input8:I1.0
A      Bit_1Hz:T45
EU
INCD   Symbol_61:VD3300
AENO
MOVD   Symbol_61:VD3300, VD3304
AENO
*D     +10, VD3304
AENO
DTR    VD3304, VD3308
AENO
MOVR   VD3308, Symbol_111:VD3312
/R     36000.0, Symbol_111:VD3312
Network 3
// Temps fonctionnement pompe
LDD>=  Symbol_61:VD3300, 900000000
LDN    Relais_PAC:Q0.3
A      Symbol_135:V1510.3
OLD
MOVD   0, Symbol_61:VD3300
AENO
MOVD   0, Symbol_111:VD3312
AENO
MOVD   0, Symbol_113:VD3320
AENO
MOVD   0, Symbol_116:VD3332
AENO
MOVD   0, Symbol_119:VD3344
AENO
R      Symbol_135:V1510.3, 1
Network 4
// Affichage HH:mm:ss sur IHM VD3320
LD     Bit_1:M1.0
TRUNC  Symbol_111:VD3312, Symbol_112:VD3316
AENO
DTR    Symbol_112:VD3316, Symbol_113:VD3320
Network 5
// Affichage hh:MM:ss sur IHM VD3032
LD     Bit_1:M1.0
MOVR   Symbol_111:VD3312, Symbol_114:VD3324
AENO
-R     Symbol_113:VD3320, Symbol_114:VD3324
AENO
MOVR   Symbol_114:VD3324, Symbol_115:VD3328
AENO
*R     60.0, Symbol_115:VD3328
AENO
TRUNC  Symbol_115:VD3328, Symbol_116:VD3332
AENO
DTR    Symbol_116:VD3332, Symbol_117:VD3336
Network 6
// Affichage hh:mm:SS sur IHM VD3044
LD     Bit_1:M1.0
MOVR   Symbol_111:VD3312, Symbol_114:VD3324
AENO
-R     Symbol_113:VD3320, Symbol_114:VD3324
AENO
MOVR   Symbol_114:VD3324, Symbol_115:VD3328
AENO
*R     60.0, Symbol_115:VD3328
AENO
TRUNC  Symbol_115:VD3328, Symbol_116:VD3332
AENO
DTR    Symbol_116:VD3332, Symbol_117:VD3336
Network 9
// Titre de réseau
// Commentaire de réseau
END_SUBROUTINE_BLOCK

SUBROUTINE_BLOCK Gestion_pH:SBR4
TITLE=Subroutine Comments
BEGIN
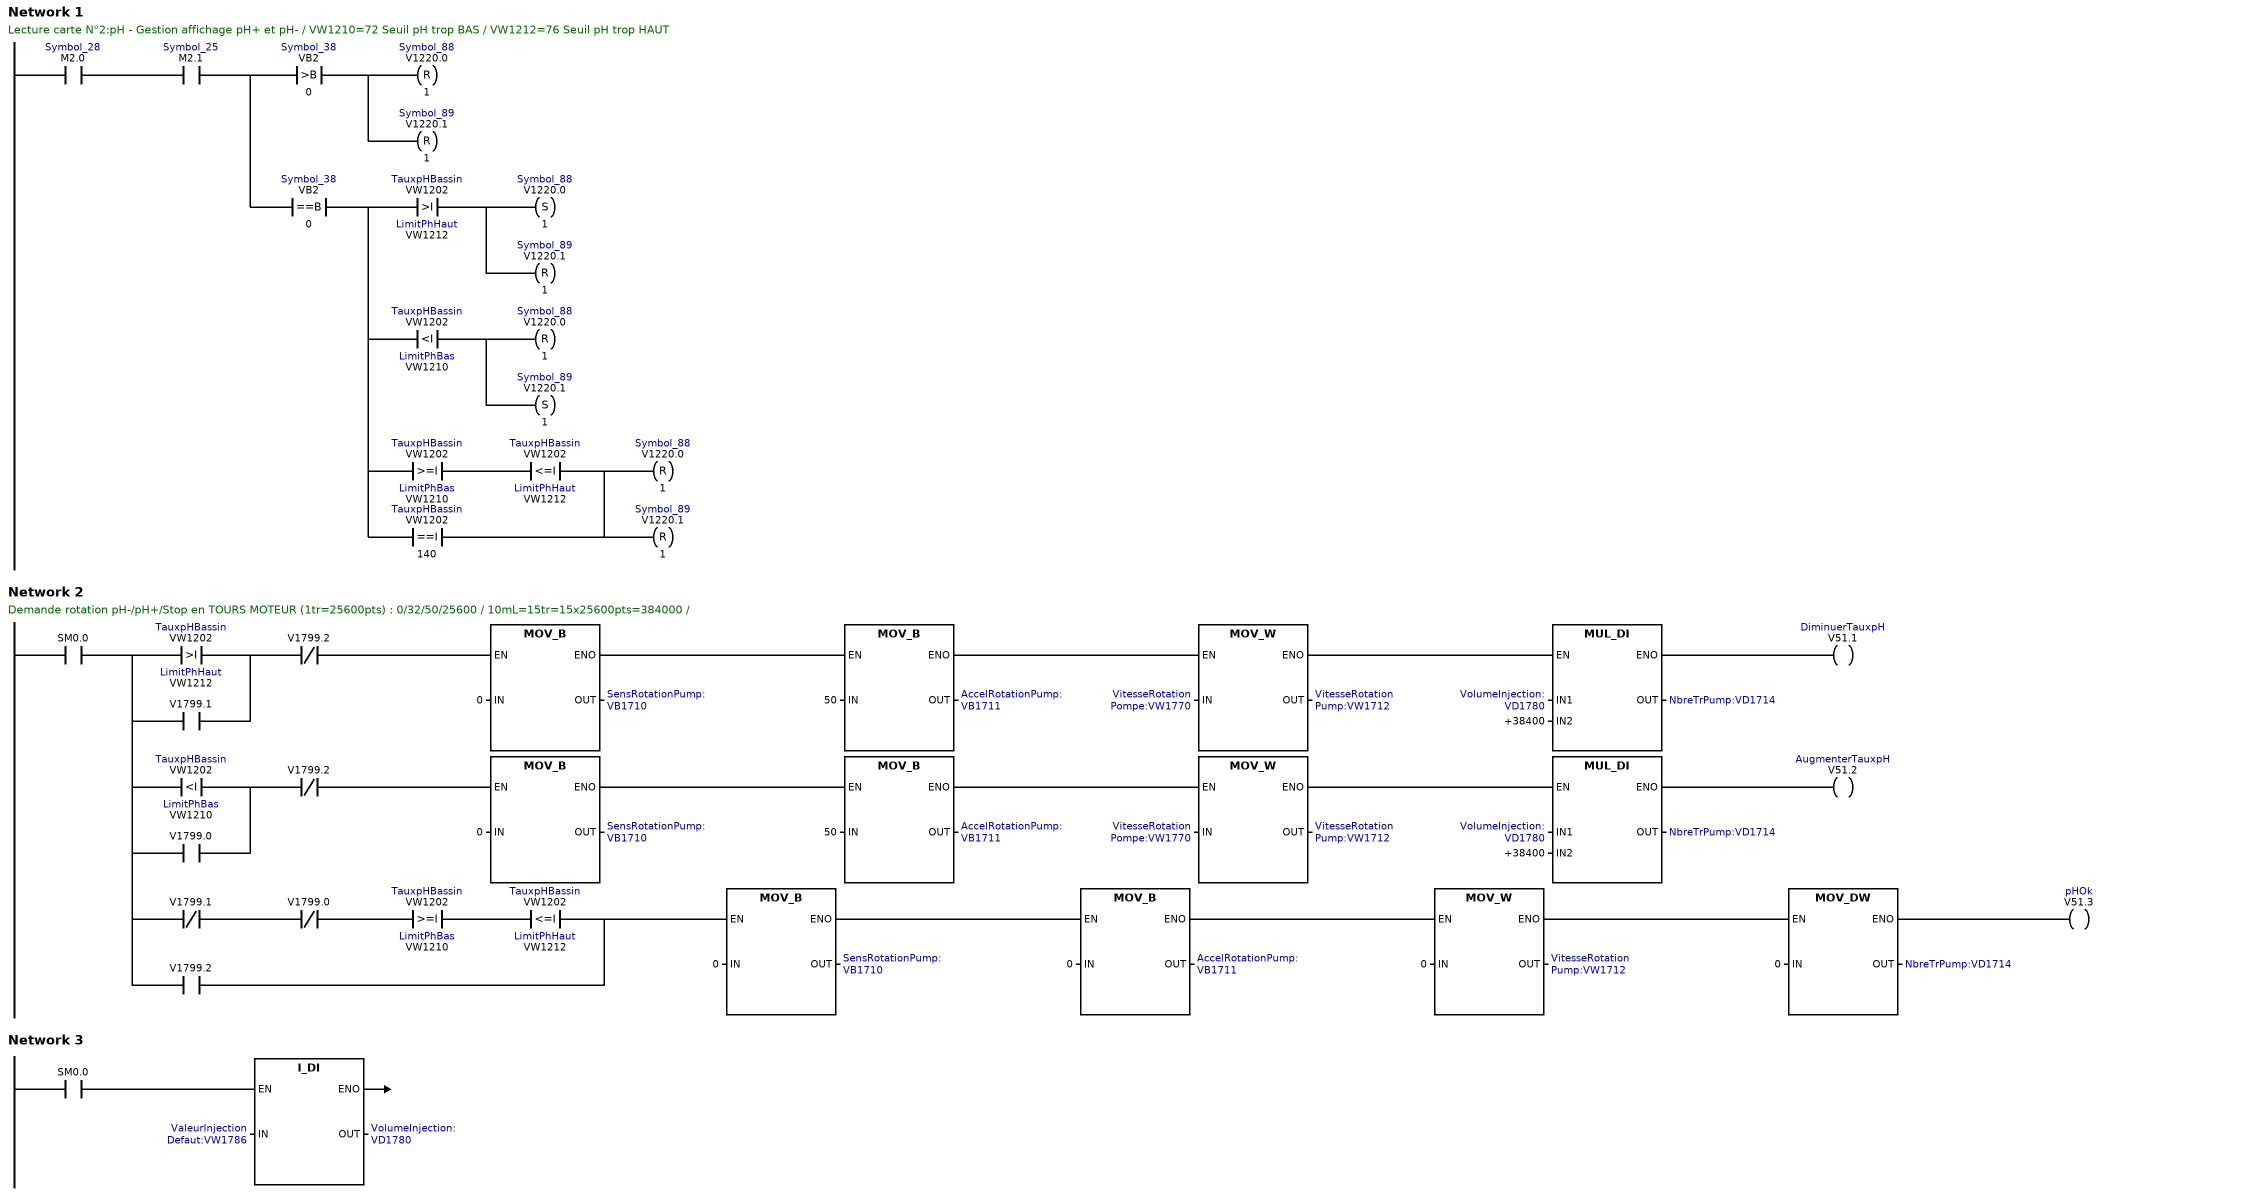
Network 1
// Lecture carte N°2:pH - Gestion affichage pH+ et pH-
// VW1210=72 Seuil pH trop BAS
// VW1212=76 Seuil pH trop HAUT
LD     Symbol_28:M2.0
A      Symbol_25:M2.1
LPS
AB>    Symbol_38:VB2, 0
R      Symbol_88:V1220.0, 1
R      Symbol_89:V1220.1, 1
LPP
AB=    Symbol_38:VB2, 0
LPS
AW>    TauxpHBassin:VW1202, LimitPhHaut:VW1212
S      Symbol_88:V1220.0, 1
R      Symbol_89:V1220.1, 1
LRD
AW<    TauxpHBassin:VW1202, LimitPhBas:VW1210
R      Symbol_88:V1220.0, 1
S      Symbol_89:V1220.1, 1
LPP
LDW>=  TauxpHBassin:VW1202, LimitPhBas:VW1210
AW<=   TauxpHBassin:VW1202, LimitPhHaut:VW1212
OW=    TauxpHBassin:VW1202, 140
ALD
R      Symbol_88:V1220.0, 1
R      Symbol_89:V1220.1, 1
Network 2
// Demande rotation pH-/pH+/Stop en TOURS MOTEUR (1tr=25600pts) : 0/32/50/25600
// 10mL=15tr=15x25600pts=384000
// 
LD     SM0.0
LPS
LDW>   TauxpHBassin:VW1202, LimitPhHaut:VW1212
O      V1799.1
ALD
AN     V1799.2
MOVB   0, SensRotationPump:VB1710
AENO
MOVB   50, AccelRotationPump:VB1711
AENO
MOVW   VitesseRotationPompe:VW1770, VitesseRotationPump:VW1712
AENO
MOVD   VolumeInjection:VD1780, NbreTrPump:VD1714
AENO
*D     +38400, NbreTrPump:VD1714
AENO
=      DiminuerTauxpH:V51.1
LRD
LDW<   TauxpHBassin:VW1202, LimitPhBas:VW1210
O      V1799.0
ALD
AN     V1799.2
MOVB   0, SensRotationPump:VB1710
AENO
MOVB   50, AccelRotationPump:VB1711
AENO
MOVW   VitesseRotationPompe:VW1770, VitesseRotationPump:VW1712
AENO
MOVD   VolumeInjection:VD1780, NbreTrPump:VD1714
AENO
*D     +38400, NbreTrPump:VD1714
AENO
=      AugmenterTauxpH:V51.2
LPP
LDN    V1799.1
AN     V1799.0
AW>=   TauxpHBassin:VW1202, LimitPhBas:VW1210
AW<=   TauxpHBassin:VW1202, LimitPhHaut:VW1212
O      V1799.2
ALD
MOVB   0, SensRotationPump:VB1710
AENO
MOVB   0, AccelRotationPump:VB1711
AENO
MOVW   0, VitesseRotationPump:VW1712
AENO
MOVD   0, NbreTrPump:VD1714
AENO
=      pHOk:V51.3
Network 3
LD     SM0.0
ITD    ValeurInjectionDefaut:VW1786, VolumeInjection:VD1780
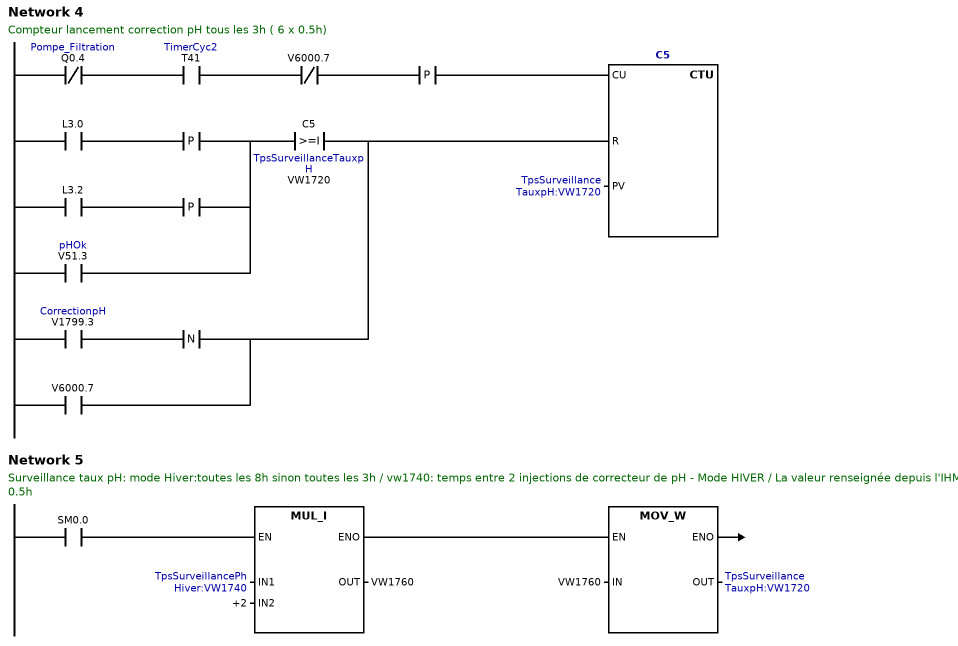
Network 4
// Compteur lancement correction pH tous les 3h ( 6 x 0.5h)
LDN    Pompe_Filtration:Q0.4
A      TimerCyc2:T41
AN     V6000.7
EU
LD     L3.0
EU
LD     L3.2
EU
OLD
O      pHOk:V51.3
AW>=   C5, TpsSurveillanceTauxpH:VW1720
LD     CorrectionpH:V1799.3
ED
O      V6000.7
OLD
CTU    C5, TpsSurveillanceTauxpH:VW1720
Network 5
// Surveillance taux pH: mode Hiver:toutes les 8h sinon toutes les 3h
// vw1740: temps entre 2 injections de correcteur de pH - Mode HIVER
// La valeur renseignée depuis l'IHM est x2 car je compte les 0.5h
LD     SM0.0
MOVW   TpsSurveillancePhHiver:VW1740, VW1760
AENO
*I     +2, VW1760
AENO
MOVW   VW1760, TpsSurveillanceTauxpH:VW1720
END_SUBROUTINE_BLOCK

SUBROUTINE_BLOCK ModBUS_RS485:SBR5
TITLE=COMMENTAIRES DE SOUS-PROGRAMME
BEGIN
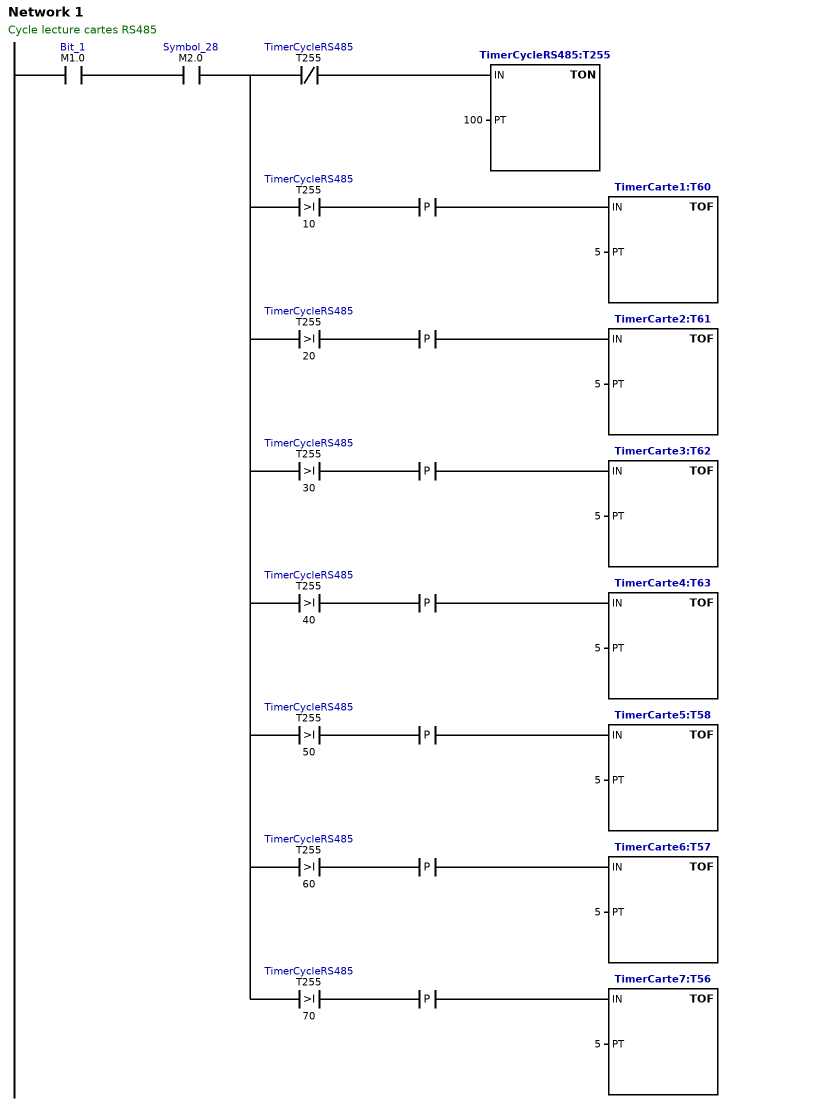
Network 1
// Cycle lecture cartes RS485
LD     Bit_1:M1.0
A      Symbol_28:M2.0
LPS
AN     TimerCycleRS485:T255
TON    TimerCycleRS485:T255, 100
LRD
AW>    TimerCycleRS485:T255, 10
EU
TOF    TimerCarte1:T60, 5
LRD
AW>    TimerCycleRS485:T255, 20
EU
TOF    TimerCarte2:T61, 5
LRD
AW>    TimerCycleRS485:T255, 30
EU
TOF    TimerCarte3:T62, 5
LRD
AW>    TimerCycleRS485:T255, 40
EU
TOF    TimerCarte4:T63, 5
LRD
AW>    TimerCycleRS485:T255, 50
EU
TOF    TimerCarte5:T58, 5
LRD
AW>    TimerCycleRS485:T255, 60
EU
TOF    TimerCarte6:T57, 5
LPP
AW>    TimerCycleRS485:T255, 70
EU
TOF    TimerCarte7:T56, 5
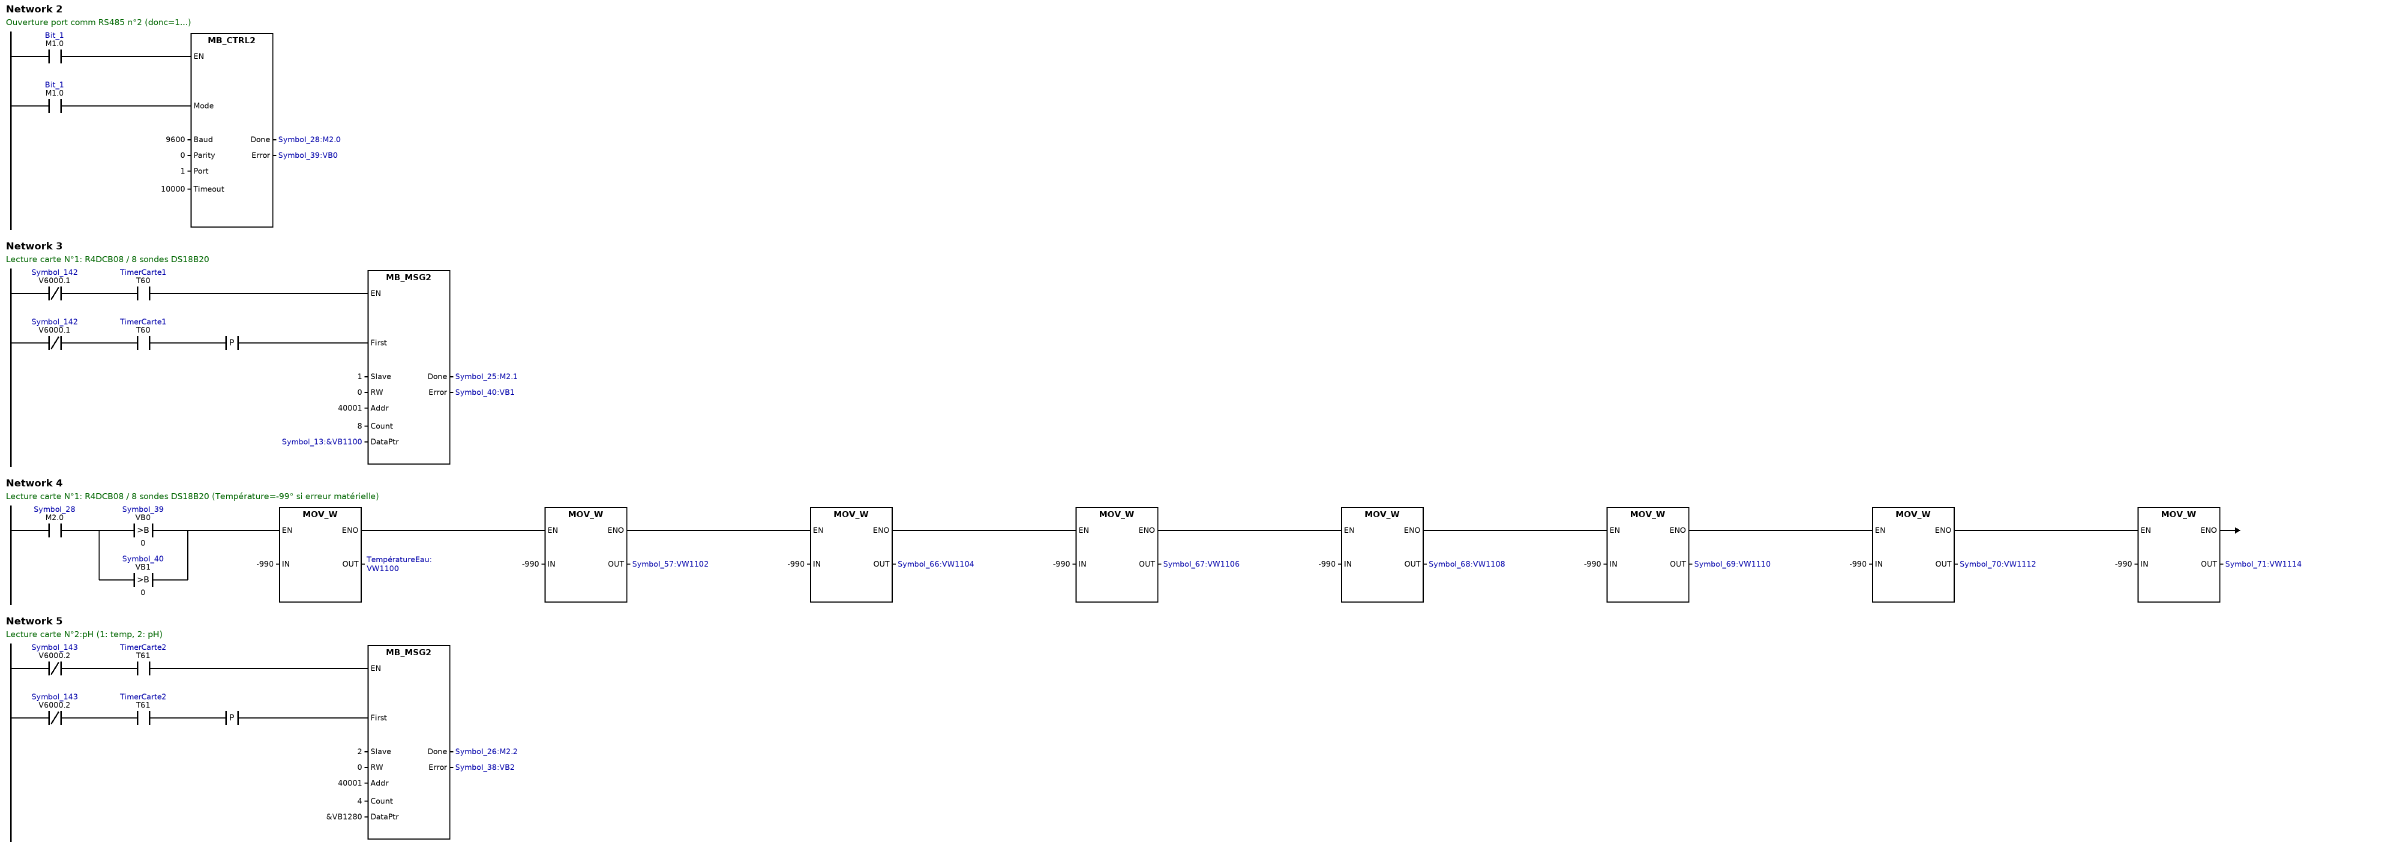
Network 2
// Ouverture port comm RS485 n°2 (donc=1...)
LD     Bit_1:M1.0
=      L60.0
LD     Bit_1:M1.0
=      L63.7
LD     L60.0
CALL   MB_CTRL2:SBR11, L63.7, 9600, 0, 1, 10000, Symbol_28:M2.0, Symbol_39:VB0
Network 3
// Lecture carte N°1: R4DCB08 / 8 sondes DS18B20
LDN    Symbol_142:V6000.1
A      TimerCarte1:T60
=      L60.0
LDN    Symbol_142:V6000.1
A      TimerCarte1:T60
EU
=      L63.7
LD     L60.0
CALL   MB_MSG2:SBR12, L63.7, 1, 0, 40001, 8, &Symbol_13:VB1100, Symbol_25:M2.1, Symbol_40:VB1
Network 4
// Lecture carte N°1: R4DCB08 / 8 sondes DS18B20 (Température=-99° si erreur matérielle)
LD     Symbol_28:M2.0
LDB>   Symbol_39:VB0, 0
OB>    Symbol_40:VB1, 0
ALD
MOVW   -990, TempératureEau:VW1100
AENO
MOVW   -990, Symbol_57:VW1102
AENO
MOVW   -990, Symbol_66:VW1104
AENO
MOVW   -990, Symbol_67:VW1106
AENO
MOVW   -990, Symbol_68:VW1108
AENO
MOVW   -990, Symbol_69:VW1110
AENO
MOVW   -990, Symbol_70:VW1112
AENO
MOVW   -990, Symbol_71:VW1114
Network 5
// Lecture carte N°2:pH (1: temp, 2: pH)
LDN    Symbol_143:V6000.2
A      TimerCarte2:T61
=      L60.0
LDN    Symbol_143:V6000.2
A      TimerCarte2:T61
EU
=      L63.7
LD     L60.0
CALL   MB_MSG2:SBR12, L63.7, 2, 0, 40001, 4, &VB1280, Symbol_26:M2.2, Symbol_38:VB2
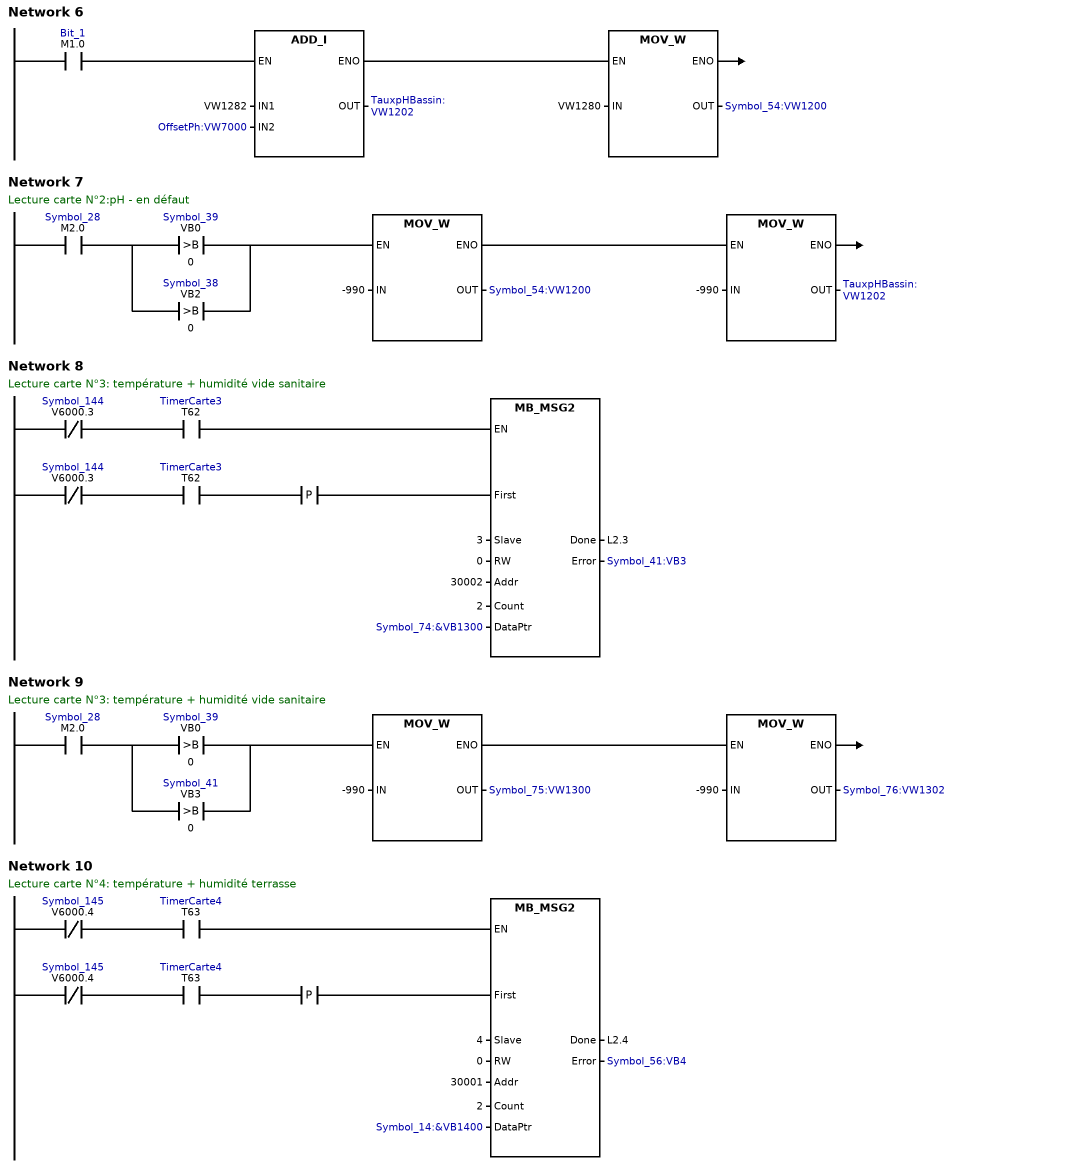
Network 6
LD     Bit_1:M1.0
MOVW   VW1282, TauxpHBassin:VW1202
AENO
+I     OffsetPh:VW7000, TauxpHBassin:VW1202
AENO
MOVW   VW1280, Symbol_54:VW1200
Network 7
// Lecture carte N°2:pH - en défaut
LD     Symbol_28:M2.0
LDB>   Symbol_39:VB0, 0
OB>    Symbol_38:VB2, 0
ALD
MOVW   -990, Symbol_54:VW1200
AENO
MOVW   -990, TauxpHBassin:VW1202
Network 8
// Lecture carte N°3: température + humidité vide sanitaire
LDN    Symbol_144:V6000.3
A      TimerCarte3:T62
=      L60.0
LDN    Symbol_144:V6000.3
A      TimerCarte3:T62
EU
=      L63.7
LD     L60.0
CALL   MB_MSG2:SBR12, L63.7, 3, 0, 30002, 2, &Symbol_74:VB1300, L2.3, Symbol_41:VB3
Network 9
// Lecture carte N°3: température + humidité vide sanitaire
LD     Symbol_28:M2.0
LDB>   Symbol_39:VB0, 0
OB>    Symbol_41:VB3, 0
ALD
MOVW   -990, Symbol_75:VW1300
AENO
MOVW   -990, Symbol_76:VW1302
Network 10
// Lecture carte N°4: température + humidité terrasse
LDN    Symbol_145:V6000.4
A      TimerCarte4:T63
=      L60.0
LDN    Symbol_145:V6000.4
A      TimerCarte4:T63
EU
=      L63.7
LD     L60.0
CALL   MB_MSG2:SBR12, L63.7, 4, 0, 30001, 2, &Symbol_14:VB1400, L2.4, Symbol_56:VB4
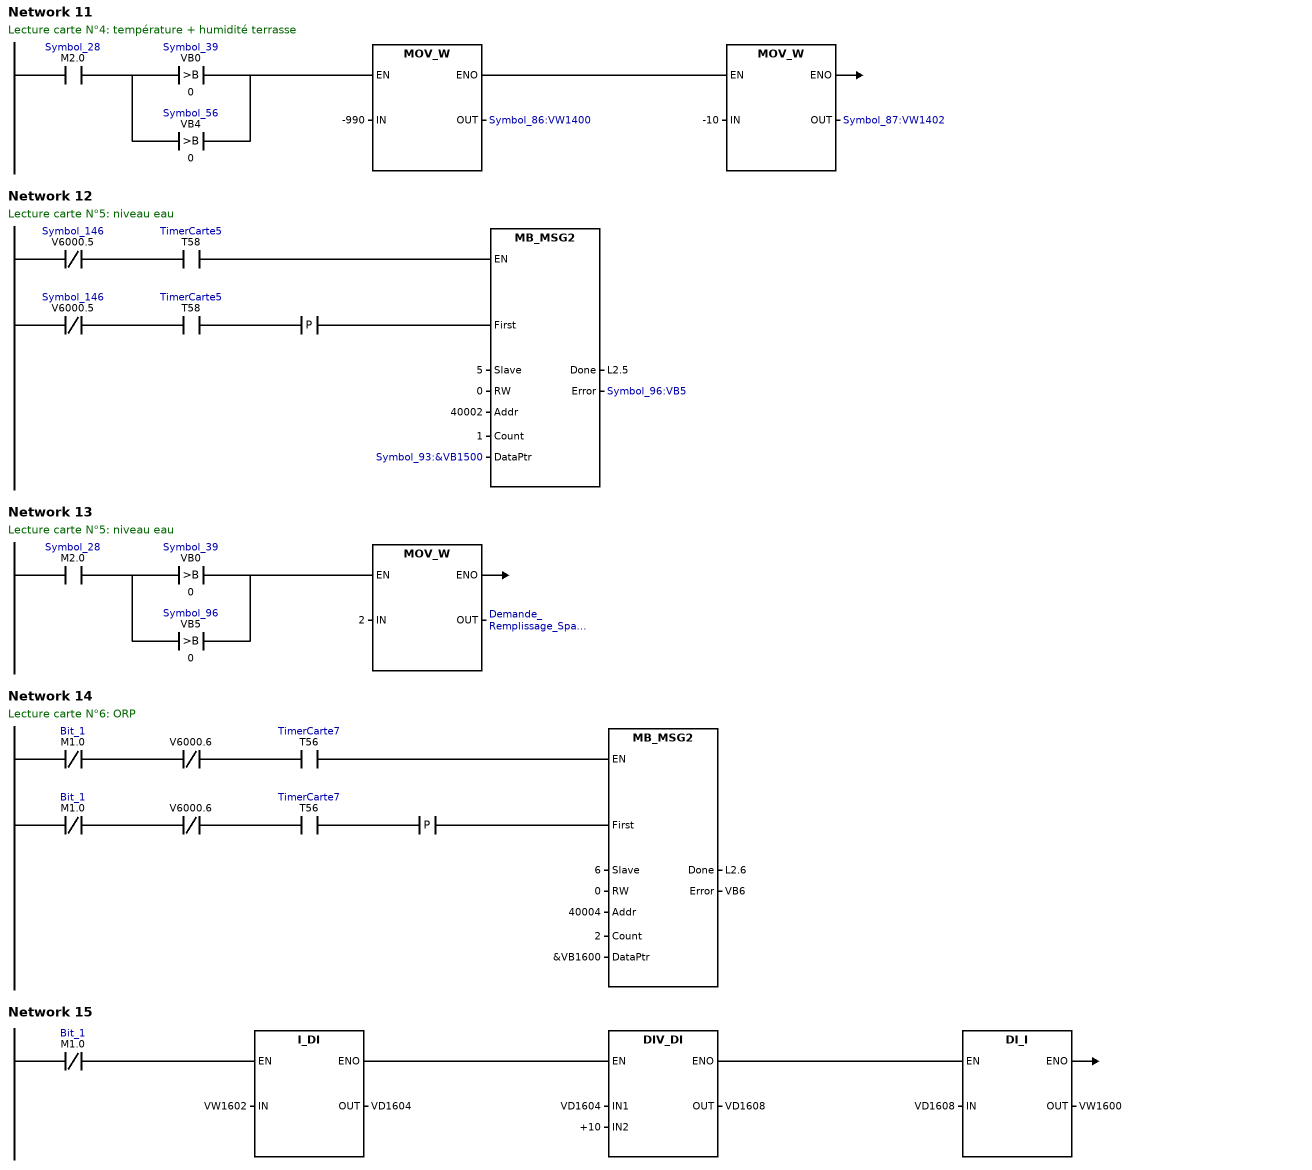
Network 11
// Lecture carte N°4: température + humidité terrasse
LD     Symbol_28:M2.0
LDB>   Symbol_39:VB0, 0
OB>    Symbol_56:VB4, 0
ALD
MOVW   -990, Symbol_86:VW1400
AENO
MOVW   -10, Symbol_87:VW1402
Network 12
// Lecture carte N°5: niveau eau
LDN    Symbol_146:V6000.5
A      TimerCarte5:T58
=      L60.0
LDN    Symbol_146:V6000.5
A      TimerCarte5:T58
EU
=      L63.7
LD     L60.0
CALL   MB_MSG2:SBR12, L63.7, 5, 0, 40002, 1, &Symbol_93:VB1500, L2.5, Symbol_96:VB5
Network 13
// Lecture carte N°5: niveau eau
LD     Symbol_28:M2.0
LDB>   Symbol_39:VB0, 0
OB>    Symbol_96:VB5, 0
ALD
MOVW   2, Demande_Remplissage_Spa:VW1520
Network 14
// Lecture carte N°6: ORP
LDN    Bit_1:M1.0
AN     V6000.6
A      TimerCarte7:T56
=      L60.0
LDN    Bit_1:M1.0
AN     V6000.6
A      TimerCarte7:T56
EU
=      L63.7
LD     L60.0
CALL   MB_MSG2:SBR12, L63.7, 6, 0, 40004, 2, &VB1600, L2.6, VB6
Network 15
LDN    Bit_1:M1.0
ITD    VW1602, VD1604
AENO
MOVD   VD1604, VD1608
AENO
/D     +10, VD1608
AENO
DTI    VD1608, VW1600
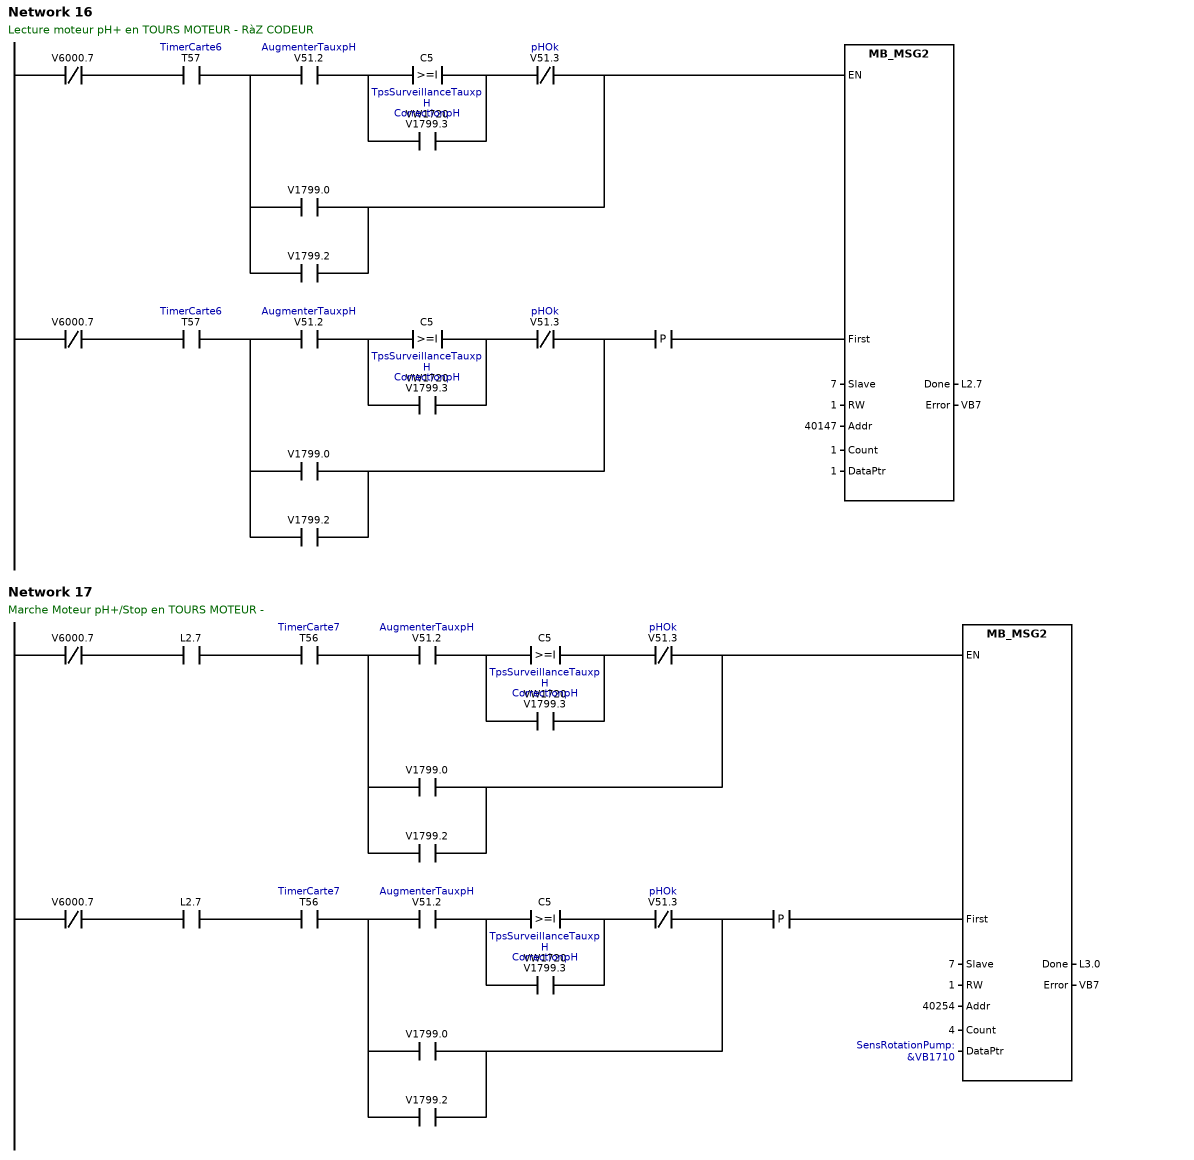
Network 16
// Lecture moteur pH+ en TOURS MOTEUR - RàZ CODEUR
LDN    V6000.7
A      TimerCarte6:T57
LD     AugmenterTauxpH:V51.2
LDW>=  C5, TpsSurveillanceTauxpH:VW1720
O      CorrectionpH:V1799.3
ALD
AN     pHOk:V51.3
LD     V1799.0
O      V1799.2
OLD
ALD
=      L60.0
LDN    V6000.7
A      TimerCarte6:T57
LD     AugmenterTauxpH:V51.2
LDW>=  C5, TpsSurveillanceTauxpH:VW1720
O      CorrectionpH:V1799.3
ALD
AN     pHOk:V51.3
LD     V1799.0
O      V1799.2
OLD
ALD
EU
=      L63.7
LD     L60.0
CALL   MB_MSG2:SBR12, L63.7, 7, 1, 40147, 1, 1, L2.7, VB7
Network 17
// Marche Moteur pH+/Stop en TOURS MOTEUR - 
LDN    V6000.7
A      L2.7
A      TimerCarte7:T56
LD     AugmenterTauxpH:V51.2
LDW>=  C5, TpsSurveillanceTauxpH:VW1720
O      CorrectionpH:V1799.3
ALD
AN     pHOk:V51.3
LD     V1799.0
O      V1799.2
OLD
ALD
=      L60.0
LDN    V6000.7
A      L2.7
A      TimerCarte7:T56
LD     AugmenterTauxpH:V51.2
LDW>=  C5, TpsSurveillanceTauxpH:VW1720
O      CorrectionpH:V1799.3
ALD
AN     pHOk:V51.3
LD     V1799.0
O      V1799.2
OLD
ALD
EU
=      L63.7
LD     L60.0
CALL   MB_MSG2:SBR12, L63.7, 7, 1, 40254, 4, &SensRotationPump:VB1710, L3.0, VB7
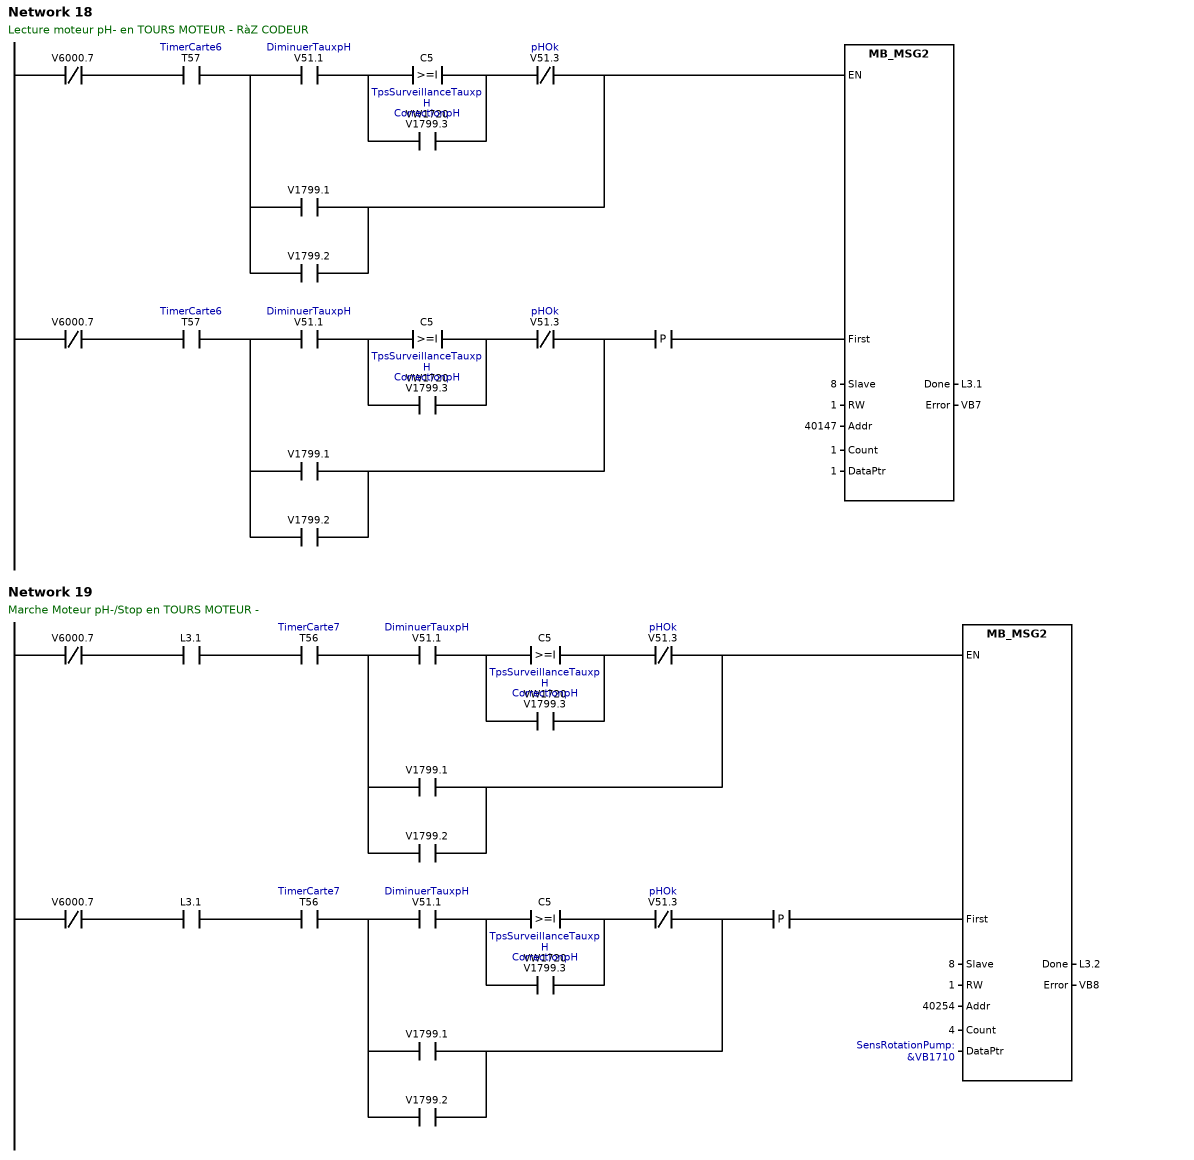
Network 18
// Lecture moteur pH- en TOURS MOTEUR - RàZ CODEUR
LDN    V6000.7
A      TimerCarte6:T57
LD     DiminuerTauxpH:V51.1
LDW>=  C5, TpsSurveillanceTauxpH:VW1720
O      CorrectionpH:V1799.3
ALD
AN     pHOk:V51.3
LD     V1799.1
O      V1799.2
OLD
ALD
=      L60.0
LDN    V6000.7
A      TimerCarte6:T57
LD     DiminuerTauxpH:V51.1
LDW>=  C5, TpsSurveillanceTauxpH:VW1720
O      CorrectionpH:V1799.3
ALD
AN     pHOk:V51.3
LD     V1799.1
O      V1799.2
OLD
ALD
EU
=      L63.7
LD     L60.0
CALL   MB_MSG2:SBR12, L63.7, 8, 1, 40147, 1, 1, L3.1, VB7
Network 19
// Marche Moteur pH-/Stop en TOURS MOTEUR - 
LDN    V6000.7
A      L3.1
A      TimerCarte7:T56
LD     DiminuerTauxpH:V51.1
LDW>=  C5, TpsSurveillanceTauxpH:VW1720
O      CorrectionpH:V1799.3
ALD
AN     pHOk:V51.3
LD     V1799.1
O      V1799.2
OLD
ALD
=      L60.0
LDN    V6000.7
A      L3.1
A      TimerCarte7:T56
LD     DiminuerTauxpH:V51.1
LDW>=  C5, TpsSurveillanceTauxpH:VW1720
O      CorrectionpH:V1799.3
ALD
AN     pHOk:V51.3
LD     V1799.1
O      V1799.2
OLD
ALD
EU
=      L63.7
LD     L60.0
CALL   MB_MSG2:SBR12, L63.7, 8, 1, 40254, 4, &SensRotationPump:VB1710, L3.2, VB8
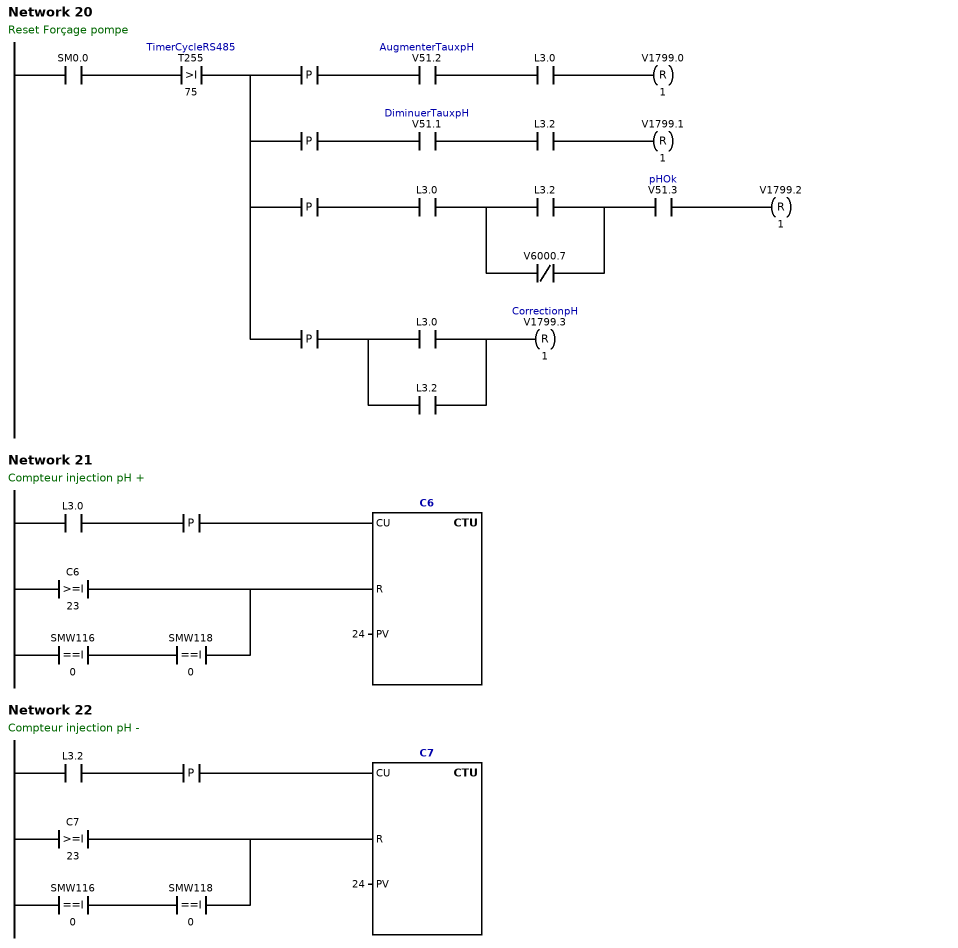
Network 20
// Reset Forçage pompe
LD     SM0.0
AW>    TimerCycleRS485:T255, 75
LPS
EU
A      AugmenterTauxpH:V51.2
A      L3.0
R      V1799.0, 1
LRD
EU
A      DiminuerTauxpH:V51.1
A      L3.2
R      V1799.1, 1
LRD
EU
A      L3.0
LD     L3.2
ON     V6000.7
ALD
A      pHOk:V51.3
R      V1799.2, 1
LPP
EU
LD     L3.0
O      L3.2
ALD
R      CorrectionpH:V1799.3, 1
Network 21
// Compteur injection pH +
LD     L3.0
EU
LDW>=  C6, 23
LDW=   SMW116, 0
AW=    SMW118, 0
OLD
CTU    C6, 24
Network 22
// Compteur injection pH -
LD     L3.2
EU
LDW>=  C7, 23
LDW=   SMW116, 0
AW=    SMW118, 0
OLD
CTU    C7, 24
END_SUBROUTINE_BLOCK

SUBROUTINE_BLOCK Gestion_Temperature:SBR6
TITLE=Subroutine Comments
BEGIN
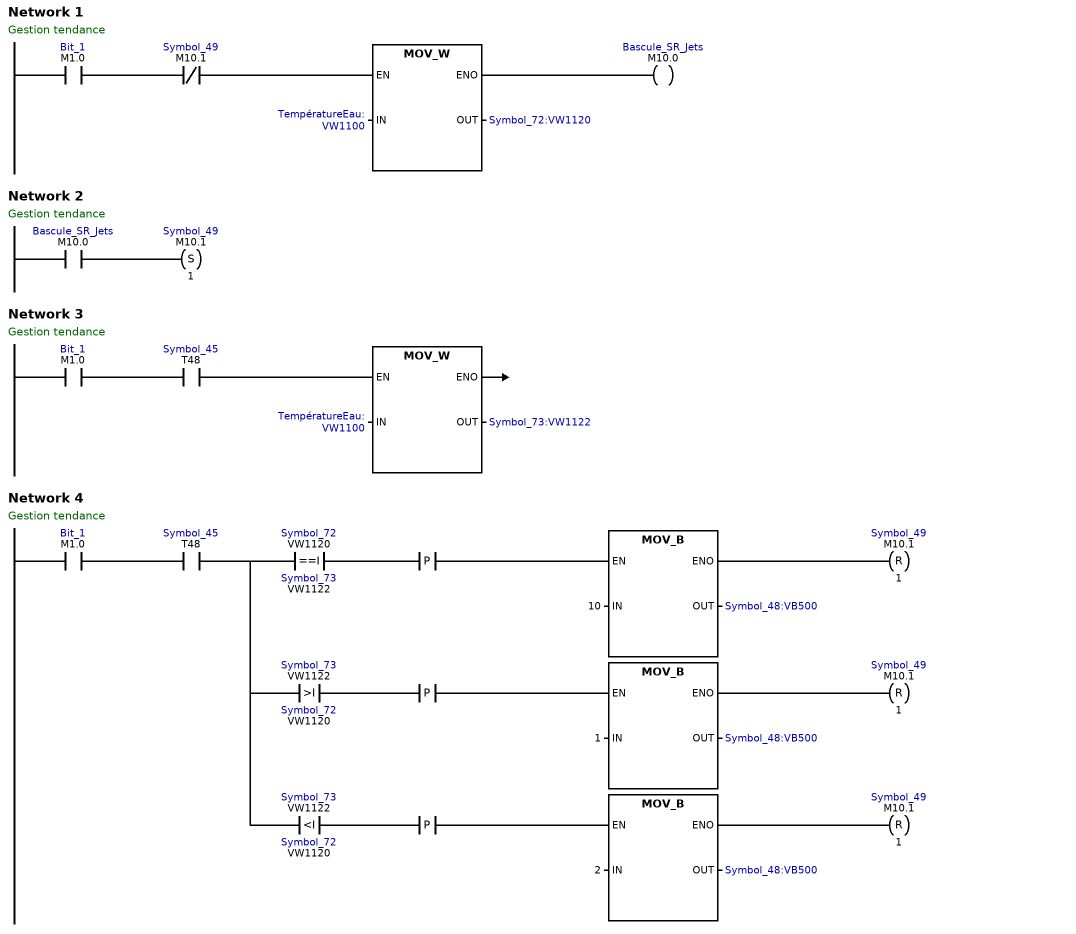
Network 1
// Gestion tendance
LD     Bit_1:M1.0
AN     Symbol_49:M10.1
MOVW   TempératureEau:VW1100, Symbol_72:VW1120
AENO
=      Bascule_SR_Jets:M10.0
Network 2
// Gestion tendance
LD     Bascule_SR_Jets:M10.0
S      Symbol_49:M10.1, 1
Network 3
// Gestion tendance
LD     Bit_1:M1.0
A      Symbol_45:T48
MOVW   TempératureEau:VW1100, Symbol_73:VW1122
Network 4
// Gestion tendance
LD     Bit_1:M1.0
A      Symbol_45:T48
LPS
AW=    Symbol_72:VW1120, Symbol_73:VW1122
EU
MOVB   10, Symbol_48:VB500
AENO
R      Symbol_49:M10.1, 1
LRD
AW>    Symbol_73:VW1122, Symbol_72:VW1120
EU
MOVB   1, Symbol_48:VB500
AENO
R      Symbol_49:M10.1, 1
LPP
AW<    Symbol_73:VW1122, Symbol_72:VW1120
EU
MOVB   2, Symbol_48:VB500
AENO
R      Symbol_49:M10.1, 1
END_SUBROUTINE_BLOCK

SUBROUTINE_BLOCK Gestion_Filtration:SBR7
TITLE=COMMENTAIRES DE SOUS-PROGRAMME
VAR
FiltReq:BOOL;	// L0.0 
END_VAR
BEGIN
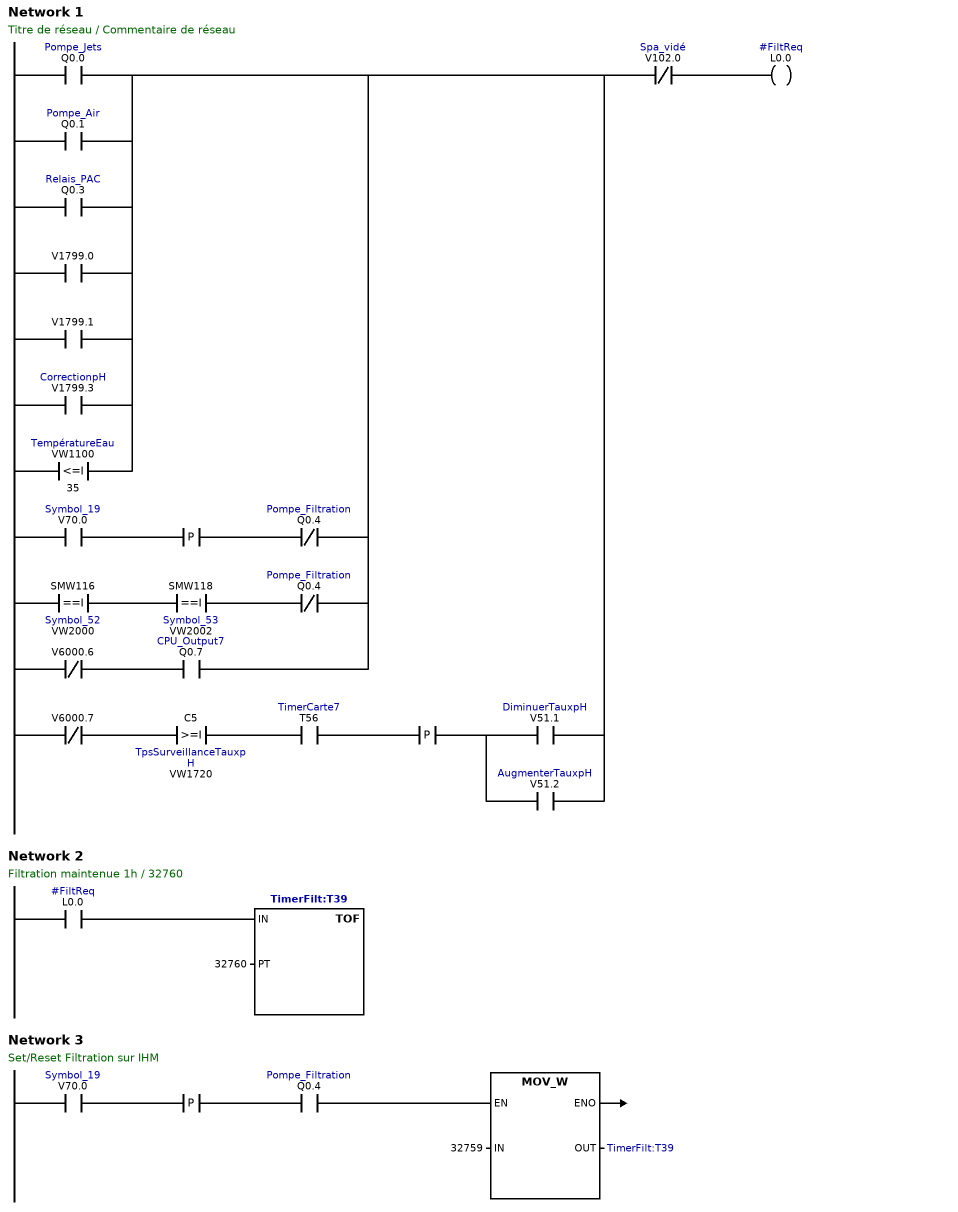
Network 1
// Titre de réseau
// Commentaire de réseau
LD     Pompe_Jets:Q0.0
O      Pompe_Air:Q0.1
O      Relais_PAC:Q0.3
O      V1799.0
O      V1799.1
O      CorrectionpH:V1799.3
OW<=   TempératureEau:VW1100, 35
LD     Symbol_19:V70.0
EU
AN     Pompe_Filtration:Q0.4
OLD
LDW=   SMW116, Symbol_52:VW2000
AW=    SMW118, Symbol_53:VW2002
AN     Pompe_Filtration:Q0.4
OLD
LDN    V6000.6
A      CPU_Output7:Q0.7
OLD
LDN    V6000.7
AW>=   C5, TpsSurveillanceTauxpH:VW1720
A      TimerCarte7:T56
EU
LD     DiminuerTauxpH:V51.1
O      AugmenterTauxpH:V51.2
ALD
OLD
AN     Spa_vidé:V102.0
=      #FiltReq:L0.0
Network 2
// Filtration maintenue 1h / 32760
LD     #FiltReq:L0.0
TOF    TimerFilt:T39, 32760
Network 3
// Set/Reset Filtration sur IHM
LD     Symbol_19:V70.0
EU
A      Pompe_Filtration:Q0.4
MOVW   32759, TimerFilt:T39
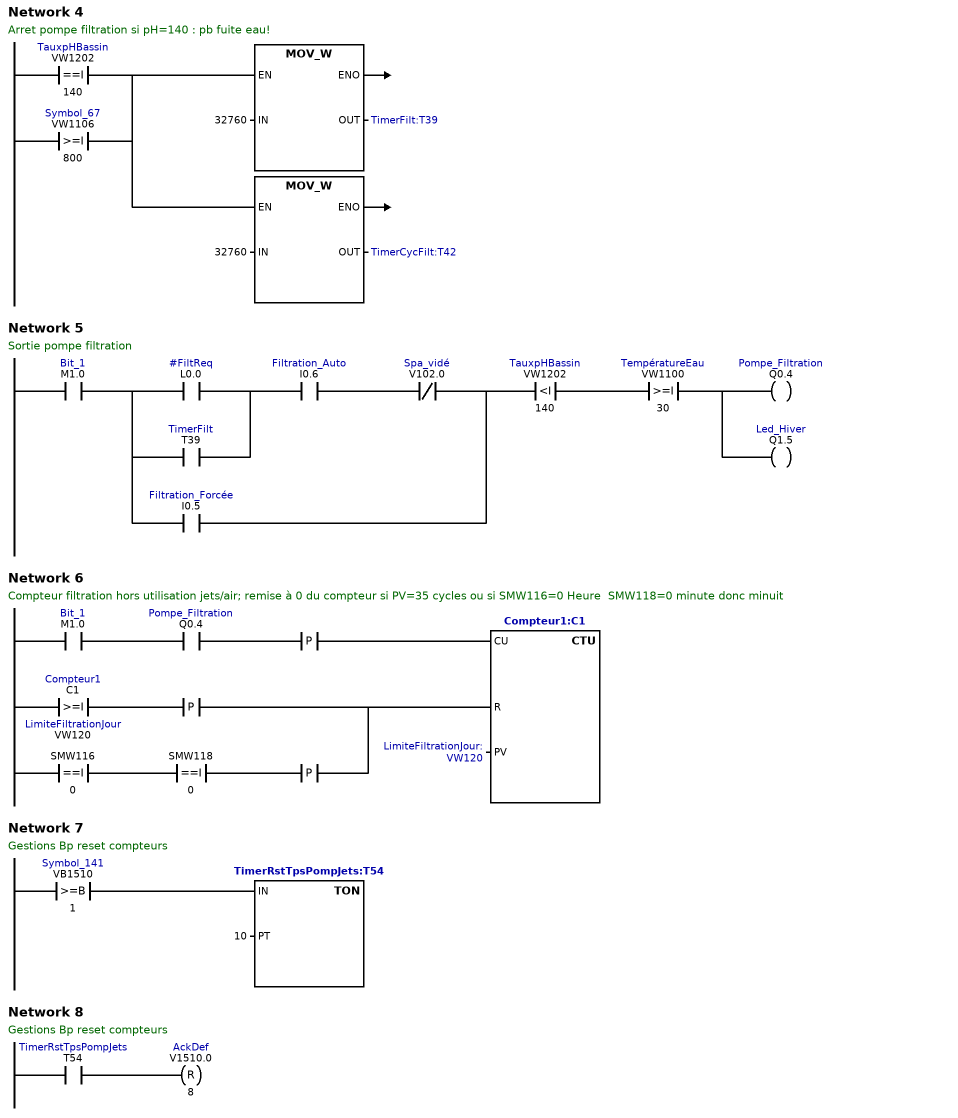
Network 4
// Arret pompe filtration si pH=140 : pb fuite eau!
LDW=   TauxpHBassin:VW1202, 140
OW>=   Symbol_67:VW1106, 800
MOVW   32760, TimerFilt:T39
MOVW   32760, TimerCycFilt:T42
Network 5
// Sortie pompe filtration
LD     Bit_1:M1.0
LD     #FiltReq:L0.0
O      TimerFilt:T39
A      Filtration_Auto:I0.6
AN     Spa_vidé:V102.0
O      Filtration_Forcée:I0.5
ALD
AW<    TauxpHBassin:VW1202, 140
AW>=   TempératureEau:VW1100, 30
=      Pompe_Filtration:Q0.4
=      Led_Hiver:Q1.5
Network 6
// Compteur filtration hors utilisation jets/air; remise à 0 du compteur si PV=35 cycles ou si SMW116=0 Heure  SMW118=0 minute donc minuit
LD     Bit_1:M1.0
A      Pompe_Filtration:Q0.4
EU
LDW>=  Compteur1:C1, LimiteFiltrationJour:VW120
EU
LDW=   SMW116, 0
AW=    SMW118, 0
EU
OLD
CTU    Compteur1:C1, LimiteFiltrationJour:VW120
Network 7
// Gestions Bp reset compteurs
LDB>=  Symbol_141:VB1510, 1
TON    TimerRstTpsPompJets:T54, 10
Network 8
// Gestions Bp reset compteurs
LD     TimerRstTpsPompJets:T54
R      AckDef:V1510.0, 8
